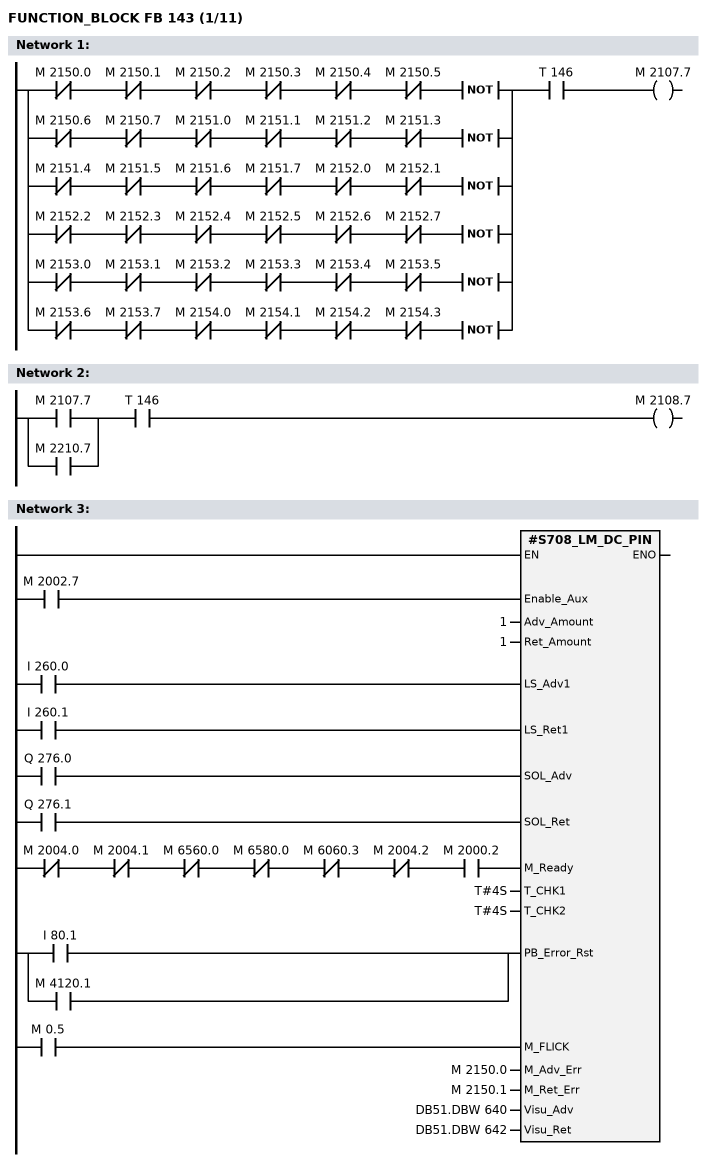

      A(    ;
      AN    M   2150.0;
      AN    M   2150.1;
      AN    M   2150.2;
      AN    M   2150.3;
      AN    M   2150.4;
      AN    M   2150.5;
      NOT   ;
      O(    ;
      AN    M   2150.6;
      AN    M   2150.7;
      AN    M   2151.0;
      AN    M   2151.1;
      AN    M   2151.2;
      AN    M   2151.3;
      NOT   ;
      )     ;
      O(    ;
      AN    M   2151.4;
      AN    M   2151.5;
      AN    M   2151.6;
      AN    M   2151.7;
      AN    M   2152.0;
      AN    M   2152.1;
      NOT   ;
      )     ;
      O(    ;
      AN    M   2152.2;
      AN    M   2152.3;
      AN    M   2152.4;
      AN    M   2152.5;
      AN    M   2152.6;
      AN    M   2152.7;
      NOT   ;
      )     ;
      O(    ;
      AN    M   2153.0;
      AN    M   2153.1;
      AN    M   2153.2;
      AN    M   2153.3;
      AN    M   2153.4;
      AN    M   2153.5;
      NOT   ;
      )     ;
      O(    ;
      AN    M   2153.6;
      AN    M   2153.7;
      AN    M   2154.0;
      AN    M   2154.1;
      AN    M   2154.2;
      AN    M   2154.3;
      NOT   ;
      )     ;
      )     ;
      A     T    146;
      =     M   2107.7;
NETWORK
TITLE =

      A(    ;
      O     M   2107.7;
      O     M   2210.7;
      )     ;
      A     T    146;
      =     M   2108.7;
NETWORK
TITLE =

      A     M   2002.7;
      =     L      0.0;
      BLD   103;
      A     I    260.0;
      =     L      0.1;
      BLD   103;
      A     I    260.1;
      =     L      0.2;
      BLD   103;
      A     Q    276.0;
      =     L      1.1;
      BLD   103;
      A     Q    276.1;
      =     L      1.2;
      BLD   103;
      AN    M   2004.0;
      AN    M   2004.1;
      AN    M   6560.0;
      AN    M   6580.0;
      AN    M   6060.3;
      AN    M   2004.2;
      A     M   2000.2;
      =     L      1.3;
      BLD   103;
      A(    ;
      O     I     80.1;
      O     M   4120.1;
      )     ;
      =     L      1.5;
      BLD   103;
      A     M      0.5;
      =     L      1.6;
      BLD   103;
      CALL #S708_LM_DC_PIN (
           Enable_Aux               := L      0.0,
           Adv_Amount               := 1,
           Ret_Amount               := 1,
           LS_Adv1                  := L      0.1,
           LS_Ret1                  := L      0.2,
           SOL_Adv                  := L      1.1,
           SOL_Ret                  := L      1.2,
           M_Ready                  := L      1.3,
           T_CHK1                   := T#4S,
           T_CHK2                   := T#4S,
           PB_Error_Rst             := L      1.5,
           M_FLICK                  := L      1.6,
           M_Adv_Err                := M   2150.0,
           M_Ret_Err                := M   2150.1,
           Visu_Adv                 := DB51.DBW  640,
           Visu_Ret                 := DB51.DBW  642);
      NOP   0;
NETWORK
TITLE =
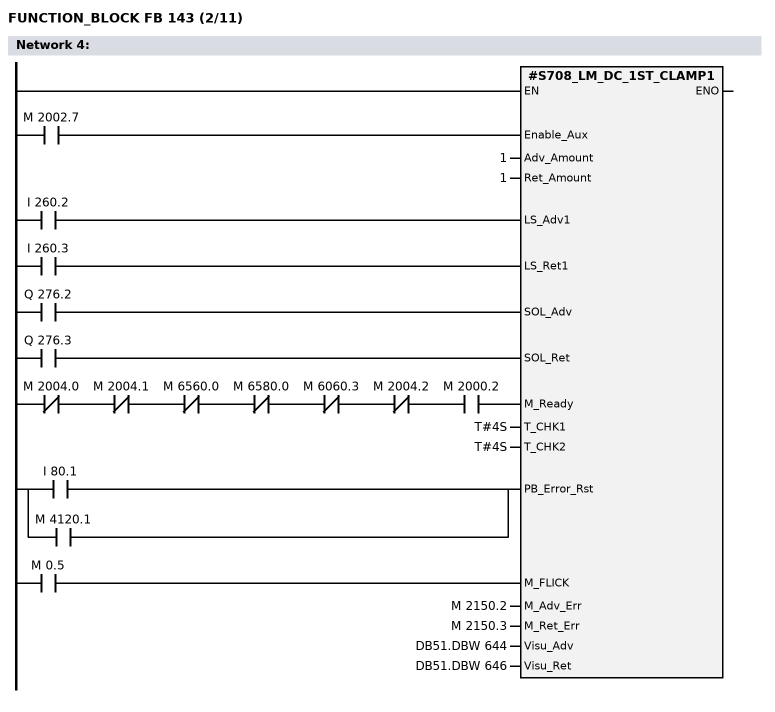

      A     M   2002.7;
      =     L      0.0;
      BLD   103;
      A     I    260.2;
      =     L      0.1;
      BLD   103;
      A     I    260.3;
      =     L      0.2;
      BLD   103;
      A     Q    276.2;
      =     L      1.1;
      BLD   103;
      A     Q    276.3;
      =     L      1.2;
      BLD   103;
      AN    M   2004.0;
      AN    M   2004.1;
      AN    M   6560.0;
      AN    M   6580.0;
      AN    M   6060.3;
      AN    M   2004.2;
      A     M   2000.2;
      =     L      1.3;
      BLD   103;
      A(    ;
      O     I     80.1;
      O     M   4120.1;
      )     ;
      =     L      1.5;
      BLD   103;
      A     M      0.5;
      =     L      1.6;
      BLD   103;
      CALL #S708_LM_DC_1ST_CLAMP1 (
           Enable_Aux               := L      0.0,
           Adv_Amount               := 1,
           Ret_Amount               := 1,
           LS_Adv1                  := L      0.1,
           LS_Ret1                  := L      0.2,
           SOL_Adv                  := L      1.1,
           SOL_Ret                  := L      1.2,
           M_Ready                  := L      1.3,
           T_CHK1                   := T#4S,
           T_CHK2                   := T#4S,
           PB_Error_Rst             := L      1.5,
           M_FLICK                  := L      1.6,
           M_Adv_Err                := M   2150.2,
           M_Ret_Err                := M   2150.3,
           Visu_Adv                 := DB51.DBW  644,
           Visu_Ret                 := DB51.DBW  646);
      NOP   0;
NETWORK
TITLE =
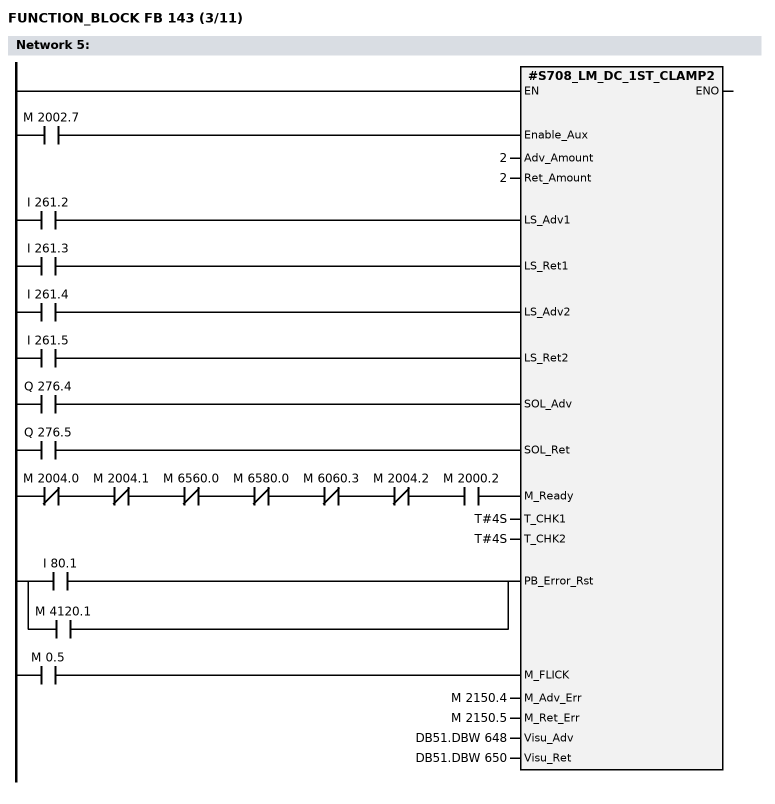

      A     M   2002.7;
      =     L      0.0;
      BLD   103;
      A     I    261.2;
      =     L      0.1;
      BLD   103;
      A     I    261.3;
      =     L      0.2;
      BLD   103;
      A     I    261.4;
      =     L      0.3;
      BLD   103;
      A     I    261.5;
      =     L      0.4;
      BLD   103;
      A     Q    276.4;
      =     L      1.1;
      BLD   103;
      A     Q    276.5;
      =     L      1.2;
      BLD   103;
      AN    M   2004.0;
      AN    M   2004.1;
      AN    M   6560.0;
      AN    M   6580.0;
      AN    M   6060.3;
      AN    M   2004.2;
      A     M   2000.2;
      =     L      1.3;
      BLD   103;
      A(    ;
      O     I     80.1;
      O     M   4120.1;
      )     ;
      =     L      1.5;
      BLD   103;
      A     M      0.5;
      =     L      1.6;
      BLD   103;
      CALL #S708_LM_DC_1ST_CLAMP2 (
           Enable_Aux               := L      0.0,
           Adv_Amount               := 2,
           Ret_Amount               := 2,
           LS_Adv1                  := L      0.1,
           LS_Ret1                  := L      0.2,
           LS_Adv2                  := L      0.3,
           LS_Ret2                  := L      0.4,
           SOL_Adv                  := L      1.1,
           SOL_Ret                  := L      1.2,
           M_Ready                  := L      1.3,
           T_CHK1                   := T#4S,
           T_CHK2                   := T#4S,
           PB_Error_Rst             := L      1.5,
           M_FLICK                  := L      1.6,
           M_Adv_Err                := M   2150.4,
           M_Ret_Err                := M   2150.5,
           Visu_Adv                 := DB51.DBW  648,
           Visu_Ret                 := DB51.DBW  650);
      NOP   0;
NETWORK
TITLE =
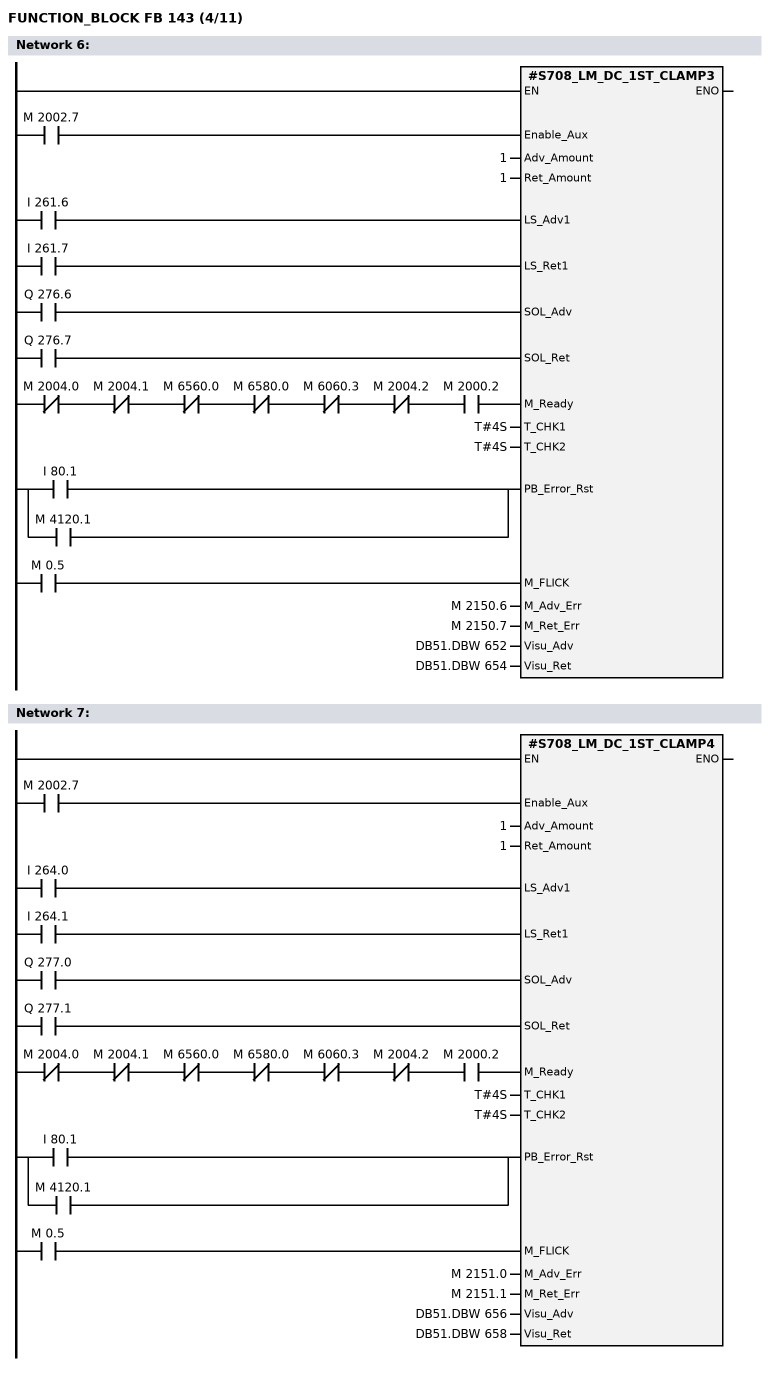

      A     M   2002.7;
      =     L      0.0;
      BLD   103;
      A     I    261.6;
      =     L      0.1;
      BLD   103;
      A     I    261.7;
      =     L      0.2;
      BLD   103;
      A     Q    276.6;
      =     L      1.1;
      BLD   103;
      A     Q    276.7;
      =     L      1.2;
      BLD   103;
      AN    M   2004.0;
      AN    M   2004.1;
      AN    M   6560.0;
      AN    M   6580.0;
      AN    M   6060.3;
      AN    M   2004.2;
      A     M   2000.2;
      =     L      1.3;
      BLD   103;
      A(    ;
      O     I     80.1;
      O     M   4120.1;
      )     ;
      =     L      1.5;
      BLD   103;
      A     M      0.5;
      =     L      1.6;
      BLD   103;
      CALL #S708_LM_DC_1ST_CLAMP3 (
           Enable_Aux               := L      0.0,
           Adv_Amount               := 1,
           Ret_Amount               := 1,
           LS_Adv1                  := L      0.1,
           LS_Ret1                  := L      0.2,
           SOL_Adv                  := L      1.1,
           SOL_Ret                  := L      1.2,
           M_Ready                  := L      1.3,
           T_CHK1                   := T#4S,
           T_CHK2                   := T#4S,
           PB_Error_Rst             := L      1.5,
           M_FLICK                  := L      1.6,
           M_Adv_Err                := M   2150.6,
           M_Ret_Err                := M   2150.7,
           Visu_Adv                 := DB51.DBW  652,
           Visu_Ret                 := DB51.DBW  654);
      NOP   0;
NETWORK
TITLE =

      A     M   2002.7;
      =     L      0.0;
      BLD   103;
      A     I    264.0;
      =     L      0.1;
      BLD   103;
      A     I    264.1;
      =     L      0.2;
      BLD   103;
      A     Q    277.0;
      =     L      1.1;
      BLD   103;
      A     Q    277.1;
      =     L      1.2;
      BLD   103;
      AN    M   2004.0;
      AN    M   2004.1;
      AN    M   6560.0;
      AN    M   6580.0;
      AN    M   6060.3;
      AN    M   2004.2;
      A     M   2000.2;
      =     L      1.3;
      BLD   103;
      A(    ;
      O     I     80.1;
      O     M   4120.1;
      )     ;
      =     L      1.5;
      BLD   103;
      A     M      0.5;
      =     L      1.6;
      BLD   103;
      CALL #S708_LM_DC_1ST_CLAMP4 (
           Enable_Aux               := L      0.0,
           Adv_Amount               := 1,
           Ret_Amount               := 1,
           LS_Adv1                  := L      0.1,
           LS_Ret1                  := L      0.2,
           SOL_Adv                  := L      1.1,
           SOL_Ret                  := L      1.2,
           M_Ready                  := L      1.3,
           T_CHK1                   := T#4S,
           T_CHK2                   := T#4S,
           PB_Error_Rst             := L      1.5,
           M_FLICK                  := L      1.6,
           M_Adv_Err                := M   2151.0,
           M_Ret_Err                := M   2151.1,
           Visu_Adv                 := DB51.DBW  656,
           Visu_Ret                 := DB51.DBW  658);
      NOP   0;
NETWORK
TITLE =
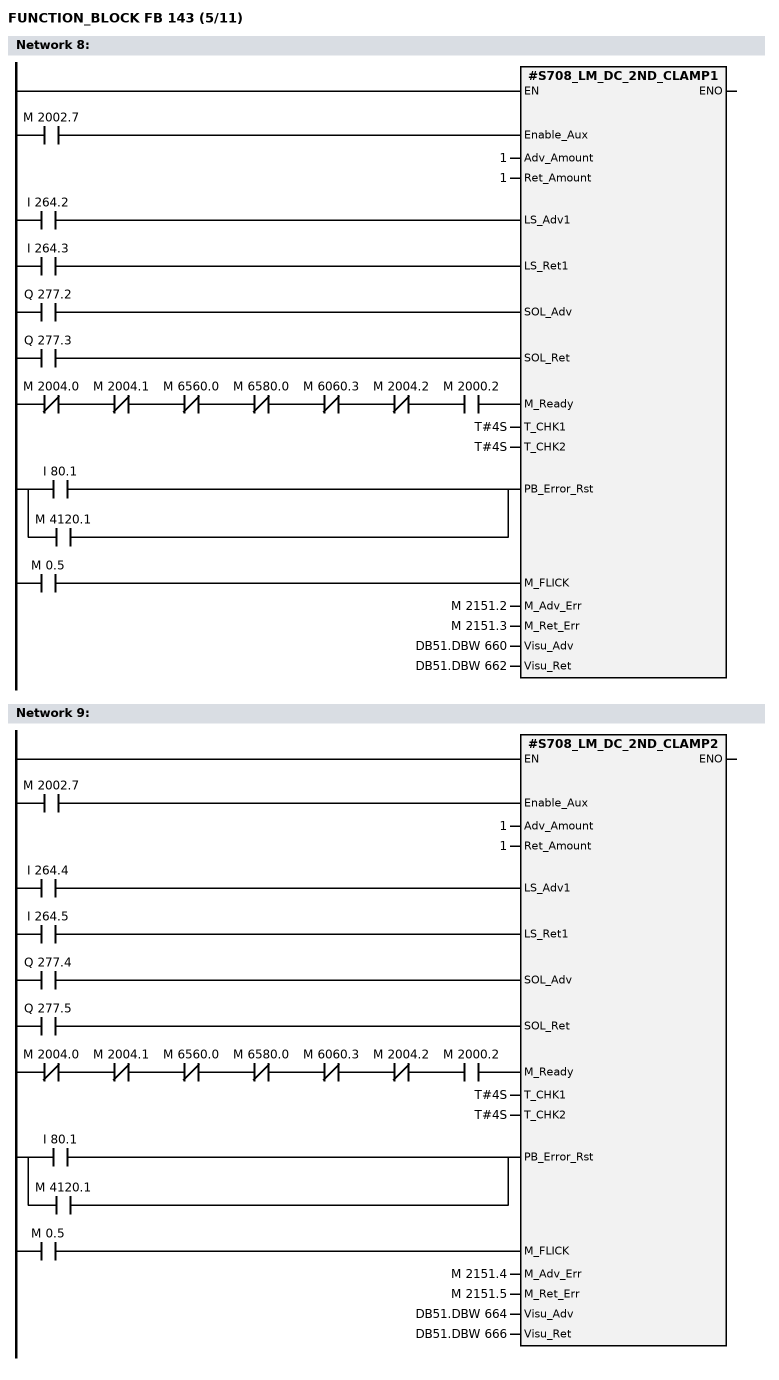

      A     M   2002.7;
      =     L      0.0;
      BLD   103;
      A     I    264.2;
      =     L      0.1;
      BLD   103;
      A     I    264.3;
      =     L      0.2;
      BLD   103;
      A     Q    277.2;
      =     L      1.1;
      BLD   103;
      A     Q    277.3;
      =     L      1.2;
      BLD   103;
      AN    M   2004.0;
      AN    M   2004.1;
      AN    M   6560.0;
      AN    M   6580.0;
      AN    M   6060.3;
      AN    M   2004.2;
      A     M   2000.2;
      =     L      1.3;
      BLD   103;
      A(    ;
      O     I     80.1;
      O     M   4120.1;
      )     ;
      =     L      1.5;
      BLD   103;
      A     M      0.5;
      =     L      1.6;
      BLD   103;
      CALL #S708_LM_DC_2ND_CLAMP1 (
           Enable_Aux               := L      0.0,
           Adv_Amount               := 1,
           Ret_Amount               := 1,
           LS_Adv1                  := L      0.1,
           LS_Ret1                  := L      0.2,
           SOL_Adv                  := L      1.1,
           SOL_Ret                  := L      1.2,
           M_Ready                  := L      1.3,
           T_CHK1                   := T#4S,
           T_CHK2                   := T#4S,
           PB_Error_Rst             := L      1.5,
           M_FLICK                  := L      1.6,
           M_Adv_Err                := M   2151.2,
           M_Ret_Err                := M   2151.3,
           Visu_Adv                 := DB51.DBW  660,
           Visu_Ret                 := DB51.DBW  662);
      NOP   0;
NETWORK
TITLE =

      A     M   2002.7;
      =     L      0.0;
      BLD   103;
      A     I    264.4;
      =     L      0.1;
      BLD   103;
      A     I    264.5;
      =     L      0.2;
      BLD   103;
      A     Q    277.4;
      =     L      1.1;
      BLD   103;
      A     Q    277.5;
      =     L      1.2;
      BLD   103;
      AN    M   2004.0;
      AN    M   2004.1;
      AN    M   6560.0;
      AN    M   6580.0;
      AN    M   6060.3;
      AN    M   2004.2;
      A     M   2000.2;
      =     L      1.3;
      BLD   103;
      A(    ;
      O     I     80.1;
      O     M   4120.1;
      )     ;
      =     L      1.5;
      BLD   103;
      A     M      0.5;
      =     L      1.6;
      BLD   103;
      CALL #S708_LM_DC_2ND_CLAMP2 (
           Enable_Aux               := L      0.0,
           Adv_Amount               := 1,
           Ret_Amount               := 1,
           LS_Adv1                  := L      0.1,
           LS_Ret1                  := L      0.2,
           SOL_Adv                  := L      1.1,
           SOL_Ret                  := L      1.2,
           M_Ready                  := L      1.3,
           T_CHK1                   := T#4S,
           T_CHK2                   := T#4S,
           PB_Error_Rst             := L      1.5,
           M_FLICK                  := L      1.6,
           M_Adv_Err                := M   2151.4,
           M_Ret_Err                := M   2151.5,
           Visu_Adv                 := DB51.DBW  664,
           Visu_Ret                 := DB51.DBW  666);
      NOP   0;
NETWORK
TITLE =
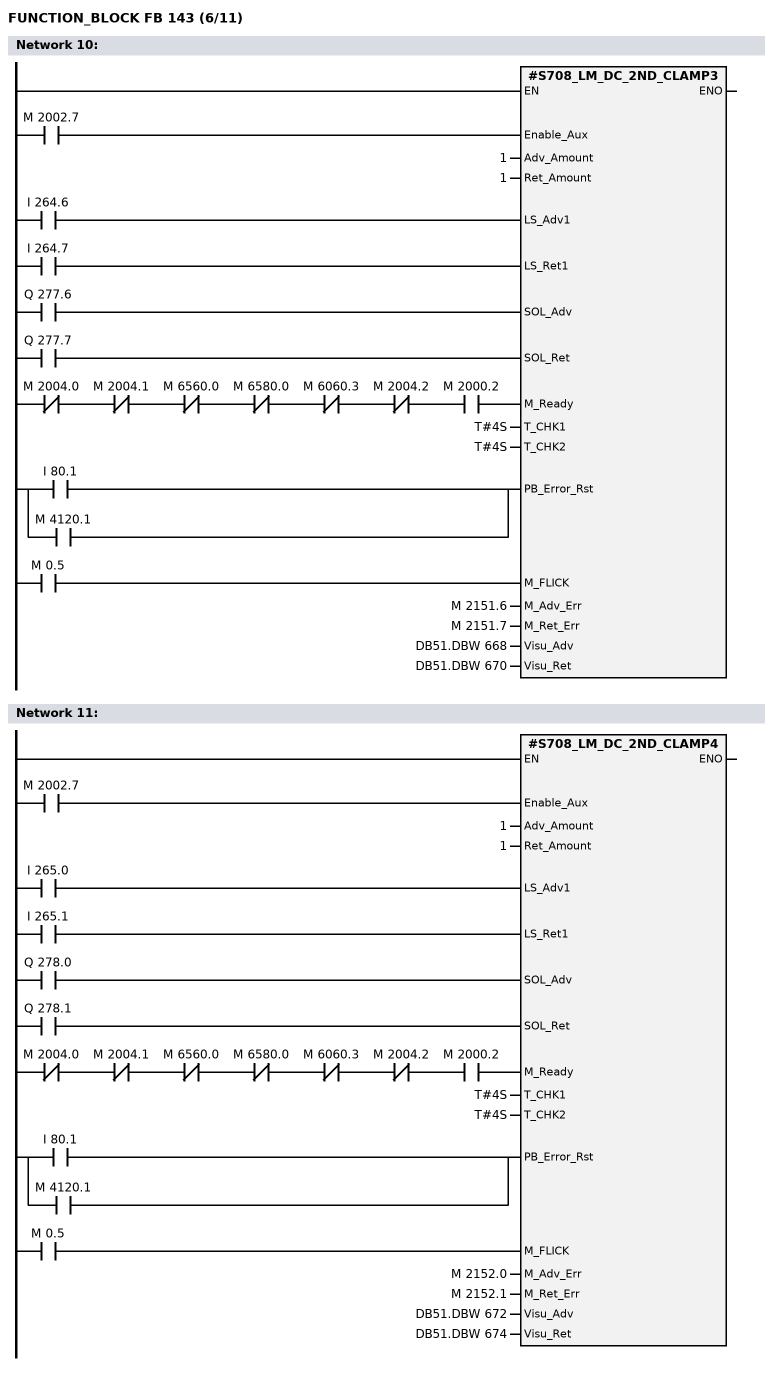

      A     M   2002.7;
      =     L      0.0;
      BLD   103;
      A     I    264.6;
      =     L      0.1;
      BLD   103;
      A     I    264.7;
      =     L      0.2;
      BLD   103;
      A     Q    277.6;
      =     L      1.1;
      BLD   103;
      A     Q    277.7;
      =     L      1.2;
      BLD   103;
      AN    M   2004.0;
      AN    M   2004.1;
      AN    M   6560.0;
      AN    M   6580.0;
      AN    M   6060.3;
      AN    M   2004.2;
      A     M   2000.2;
      =     L      1.3;
      BLD   103;
      A(    ;
      O     I     80.1;
      O     M   4120.1;
      )     ;
      =     L      1.5;
      BLD   103;
      A     M      0.5;
      =     L      1.6;
      BLD   103;
      CALL #S708_LM_DC_2ND_CLAMP3 (
           Enable_Aux               := L      0.0,
           Adv_Amount               := 1,
           Ret_Amount               := 1,
           LS_Adv1                  := L      0.1,
           LS_Ret1                  := L      0.2,
           SOL_Adv                  := L      1.1,
           SOL_Ret                  := L      1.2,
           M_Ready                  := L      1.3,
           T_CHK1                   := T#4S,
           T_CHK2                   := T#4S,
           PB_Error_Rst             := L      1.5,
           M_FLICK                  := L      1.6,
           M_Adv_Err                := M   2151.6,
           M_Ret_Err                := M   2151.7,
           Visu_Adv                 := DB51.DBW  668,
           Visu_Ret                 := DB51.DBW  670);
      NOP   0;
NETWORK
TITLE =

      A     M   2002.7;
      =     L      0.0;
      BLD   103;
      A     I    265.0;
      =     L      0.1;
      BLD   103;
      A     I    265.1;
      =     L      0.2;
      BLD   103;
      A     Q    278.0;
      =     L      1.1;
      BLD   103;
      A     Q    278.1;
      =     L      1.2;
      BLD   103;
      AN    M   2004.0;
      AN    M   2004.1;
      AN    M   6560.0;
      AN    M   6580.0;
      AN    M   6060.3;
      AN    M   2004.2;
      A     M   2000.2;
      =     L      1.3;
      BLD   103;
      A(    ;
      O     I     80.1;
      O     M   4120.1;
      )     ;
      =     L      1.5;
      BLD   103;
      A     M      0.5;
      =     L      1.6;
      BLD   103;
      CALL #S708_LM_DC_2ND_CLAMP4 (
           Enable_Aux               := L      0.0,
           Adv_Amount               := 1,
           Ret_Amount               := 1,
           LS_Adv1                  := L      0.1,
           LS_Ret1                  := L      0.2,
           SOL_Adv                  := L      1.1,
           SOL_Ret                  := L      1.2,
           M_Ready                  := L      1.3,
           T_CHK1                   := T#4S,
           T_CHK2                   := T#4S,
           PB_Error_Rst             := L      1.5,
           M_FLICK                  := L      1.6,
           M_Adv_Err                := M   2152.0,
           M_Ret_Err                := M   2152.1,
           Visu_Adv                 := DB51.DBW  672,
           Visu_Ret                 := DB51.DBW  674);
      NOP   0;
NETWORK
TITLE =
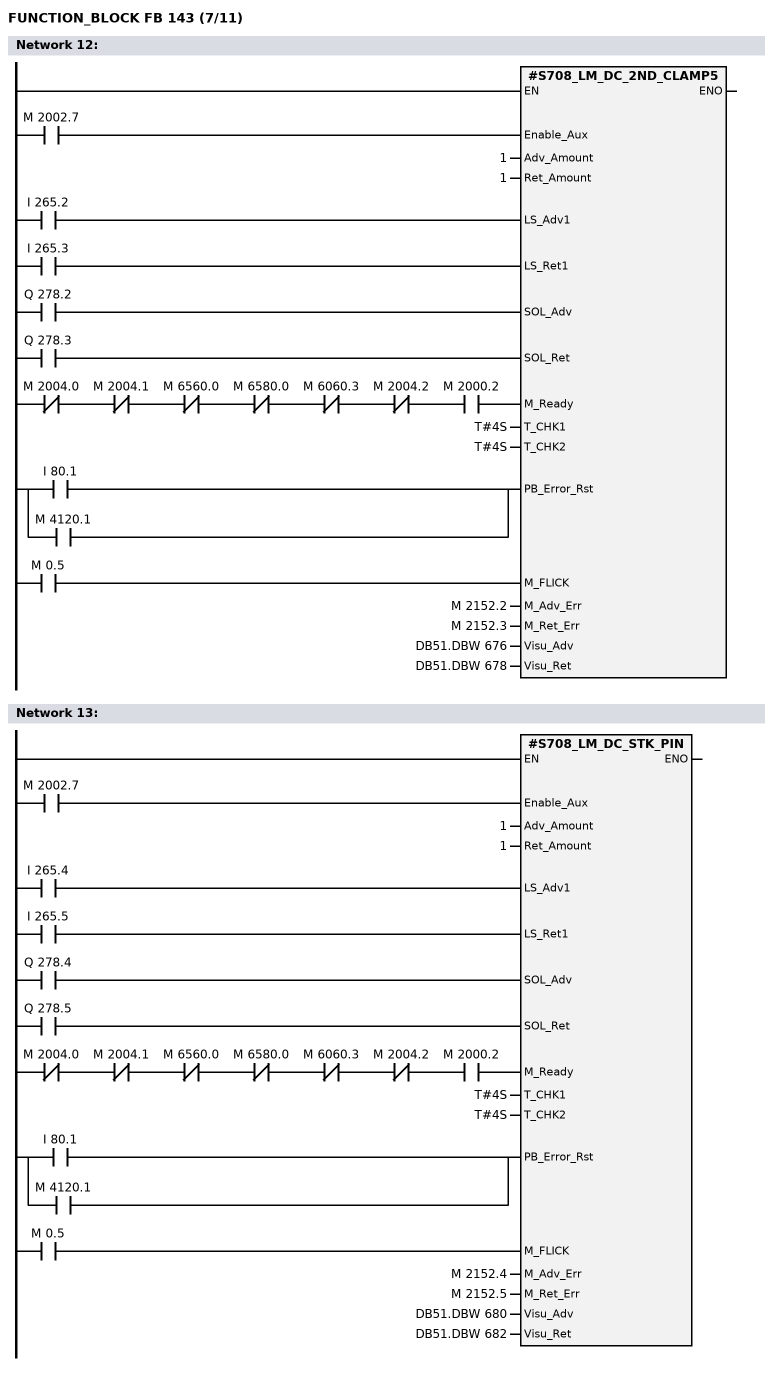

      A     M   2002.7;
      =     L      0.0;
      BLD   103;
      A     I    265.2;
      =     L      0.1;
      BLD   103;
      A     I    265.3;
      =     L      0.2;
      BLD   103;
      A     Q    278.2;
      =     L      1.1;
      BLD   103;
      A     Q    278.3;
      =     L      1.2;
      BLD   103;
      AN    M   2004.0;
      AN    M   2004.1;
      AN    M   6560.0;
      AN    M   6580.0;
      AN    M   6060.3;
      AN    M   2004.2;
      A     M   2000.2;
      =     L      1.3;
      BLD   103;
      A(    ;
      O     I     80.1;
      O     M   4120.1;
      )     ;
      =     L      1.5;
      BLD   103;
      A     M      0.5;
      =     L      1.6;
      BLD   103;
      CALL #S708_LM_DC_2ND_CLAMP5 (
           Enable_Aux               := L      0.0,
           Adv_Amount               := 1,
           Ret_Amount               := 1,
           LS_Adv1                  := L      0.1,
           LS_Ret1                  := L      0.2,
           SOL_Adv                  := L      1.1,
           SOL_Ret                  := L      1.2,
           M_Ready                  := L      1.3,
           T_CHK1                   := T#4S,
           T_CHK2                   := T#4S,
           PB_Error_Rst             := L      1.5,
           M_FLICK                  := L      1.6,
           M_Adv_Err                := M   2152.2,
           M_Ret_Err                := M   2152.3,
           Visu_Adv                 := DB51.DBW  676,
           Visu_Ret                 := DB51.DBW  678);
      NOP   0;
NETWORK
TITLE =

      A     M   2002.7;
      =     L      0.0;
      BLD   103;
      A     I    265.4;
      =     L      0.1;
      BLD   103;
      A     I    265.5;
      =     L      0.2;
      BLD   103;
      A     Q    278.4;
      =     L      1.1;
      BLD   103;
      A     Q    278.5;
      =     L      1.2;
      BLD   103;
      AN    M   2004.0;
      AN    M   2004.1;
      AN    M   6560.0;
      AN    M   6580.0;
      AN    M   6060.3;
      AN    M   2004.2;
      A     M   2000.2;
      =     L      1.3;
      BLD   103;
      A(    ;
      O     I     80.1;
      O     M   4120.1;
      )     ;
      =     L      1.5;
      BLD   103;
      A     M      0.5;
      =     L      1.6;
      BLD   103;
      CALL #S708_LM_DC_STK_PIN (
           Enable_Aux               := L      0.0,
           Adv_Amount               := 1,
           Ret_Amount               := 1,
           LS_Adv1                  := L      0.1,
           LS_Ret1                  := L      0.2,
           SOL_Adv                  := L      1.1,
           SOL_Ret                  := L      1.2,
           M_Ready                  := L      1.3,
           T_CHK1                   := T#4S,
           T_CHK2                   := T#4S,
           PB_Error_Rst             := L      1.5,
           M_FLICK                  := L      1.6,
           M_Adv_Err                := M   2152.4,
           M_Ret_Err                := M   2152.5,
           Visu_Adv                 := DB51.DBW  680,
           Visu_Ret                 := DB51.DBW  682);
      NOP   0;
NETWORK
TITLE =
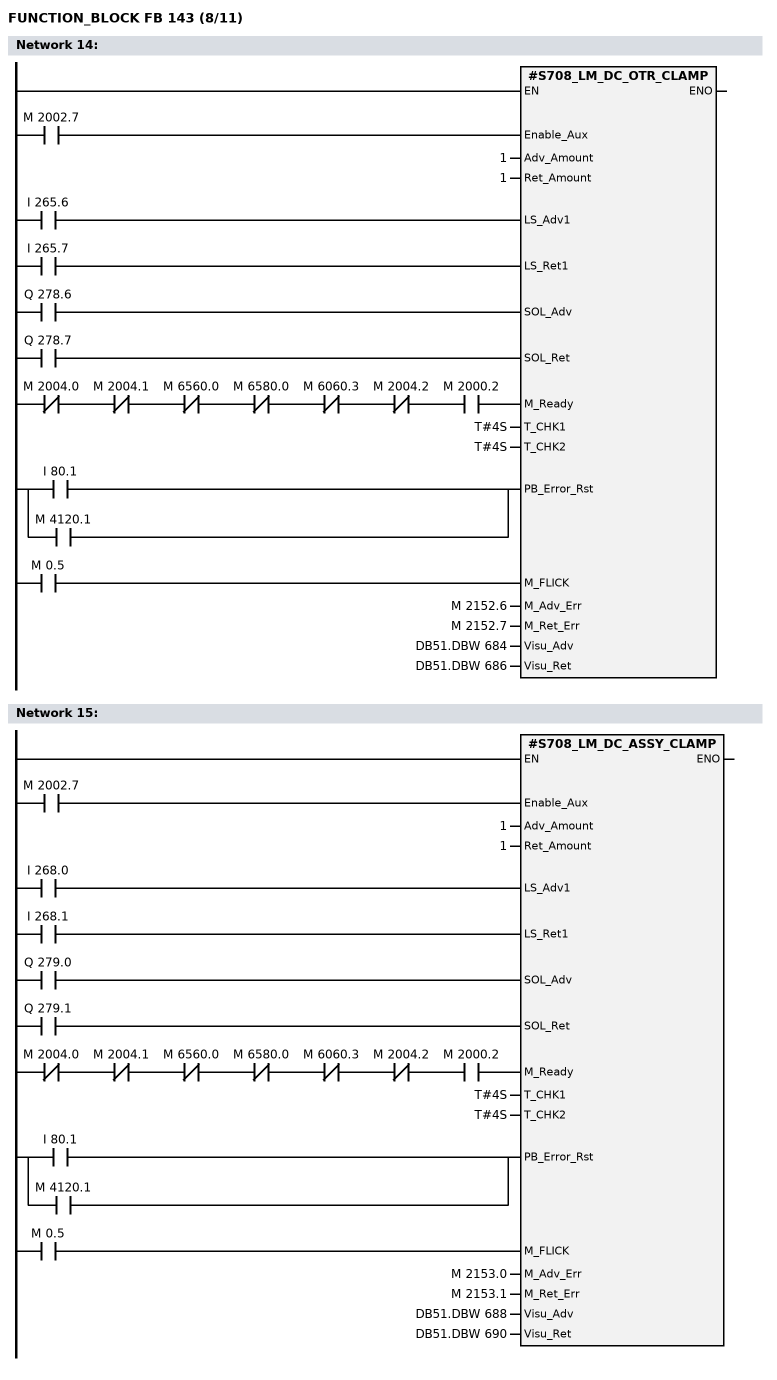

      A     M   2002.7;
      =     L      0.0;
      BLD   103;
      A     I    265.6;
      =     L      0.1;
      BLD   103;
      A     I    265.7;
      =     L      0.2;
      BLD   103;
      A     Q    278.6;
      =     L      1.1;
      BLD   103;
      A     Q    278.7;
      =     L      1.2;
      BLD   103;
      AN    M   2004.0;
      AN    M   2004.1;
      AN    M   6560.0;
      AN    M   6580.0;
      AN    M   6060.3;
      AN    M   2004.2;
      A     M   2000.2;
      =     L      1.3;
      BLD   103;
      A(    ;
      O     I     80.1;
      O     M   4120.1;
      )     ;
      =     L      1.5;
      BLD   103;
      A     M      0.5;
      =     L      1.6;
      BLD   103;
      CALL #S708_LM_DC_OTR_CLAMP (
           Enable_Aux               := L      0.0,
           Adv_Amount               := 1,
           Ret_Amount               := 1,
           LS_Adv1                  := L      0.1,
           LS_Ret1                  := L      0.2,
           SOL_Adv                  := L      1.1,
           SOL_Ret                  := L      1.2,
           M_Ready                  := L      1.3,
           T_CHK1                   := T#4S,
           T_CHK2                   := T#4S,
           PB_Error_Rst             := L      1.5,
           M_FLICK                  := L      1.6,
           M_Adv_Err                := M   2152.6,
           M_Ret_Err                := M   2152.7,
           Visu_Adv                 := DB51.DBW  684,
           Visu_Ret                 := DB51.DBW  686);
      NOP   0;
NETWORK
TITLE =

      A     M   2002.7;
      =     L      0.0;
      BLD   103;
      A     I    268.0;
      =     L      0.1;
      BLD   103;
      A     I    268.1;
      =     L      0.2;
      BLD   103;
      A     Q    279.0;
      =     L      1.1;
      BLD   103;
      A     Q    279.1;
      =     L      1.2;
      BLD   103;
      AN    M   2004.0;
      AN    M   2004.1;
      AN    M   6560.0;
      AN    M   6580.0;
      AN    M   6060.3;
      AN    M   2004.2;
      A     M   2000.2;
      =     L      1.3;
      BLD   103;
      A(    ;
      O     I     80.1;
      O     M   4120.1;
      )     ;
      =     L      1.5;
      BLD   103;
      A     M      0.5;
      =     L      1.6;
      BLD   103;
      CALL #S708_LM_DC_ASSY_CLAMP (
           Enable_Aux               := L      0.0,
           Adv_Amount               := 1,
           Ret_Amount               := 1,
           LS_Adv1                  := L      0.1,
           LS_Ret1                  := L      0.2,
           SOL_Adv                  := L      1.1,
           SOL_Ret                  := L      1.2,
           M_Ready                  := L      1.3,
           T_CHK1                   := T#4S,
           T_CHK2                   := T#4S,
           PB_Error_Rst             := L      1.5,
           M_FLICK                  := L      1.6,
           M_Adv_Err                := M   2153.0,
           M_Ret_Err                := M   2153.1,
           Visu_Adv                 := DB51.DBW  688,
           Visu_Ret                 := DB51.DBW  690);
      NOP   0;
NETWORK
TITLE =
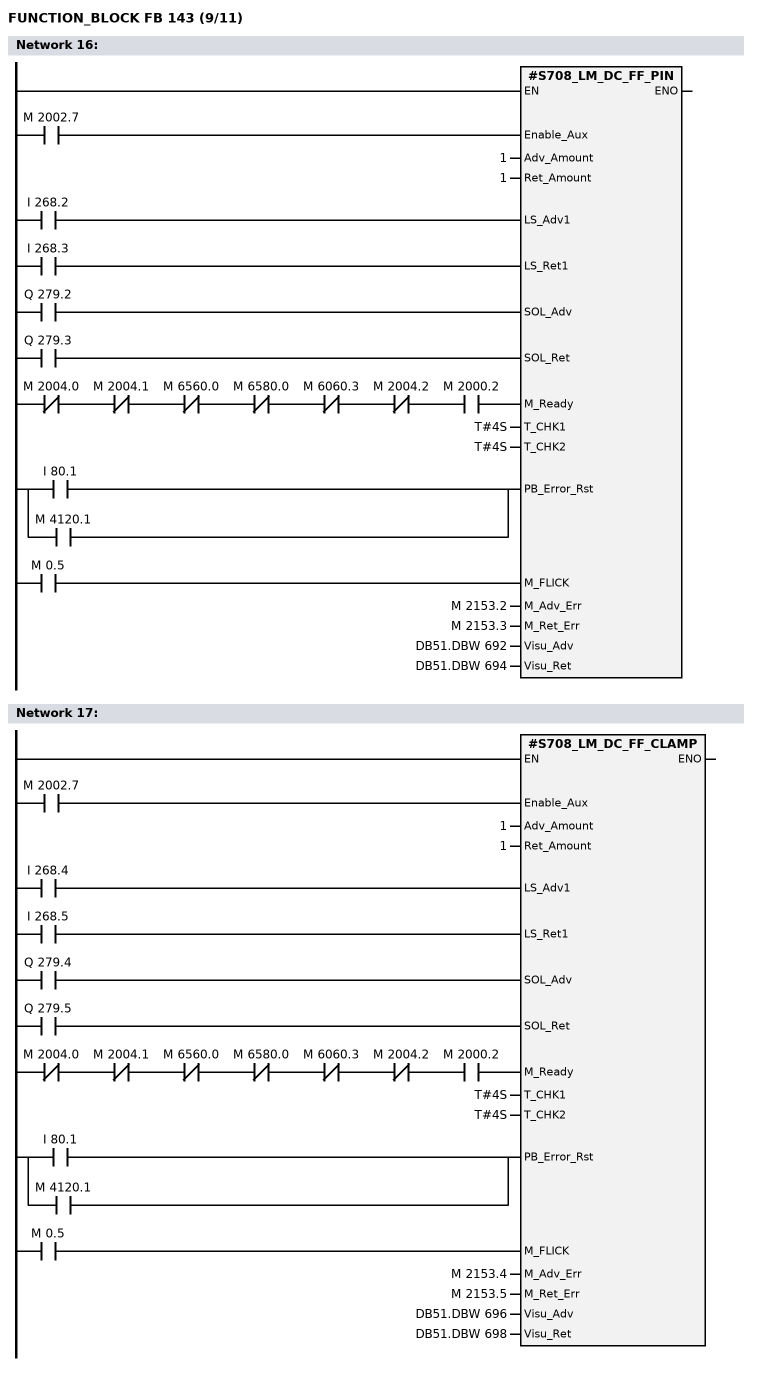

      A     M   2002.7;
      =     L      0.0;
      BLD   103;
      A     I    268.2;
      =     L      0.1;
      BLD   103;
      A     I    268.3;
      =     L      0.2;
      BLD   103;
      A     Q    279.2;
      =     L      1.1;
      BLD   103;
      A     Q    279.3;
      =     L      1.2;
      BLD   103;
      AN    M   2004.0;
      AN    M   2004.1;
      AN    M   6560.0;
      AN    M   6580.0;
      AN    M   6060.3;
      AN    M   2004.2;
      A     M   2000.2;
      =     L      1.3;
      BLD   103;
      A(    ;
      O     I     80.1;
      O     M   4120.1;
      )     ;
      =     L      1.5;
      BLD   103;
      A     M      0.5;
      =     L      1.6;
      BLD   103;
      CALL #S708_LM_DC_FF_PIN (
           Enable_Aux               := L      0.0,
           Adv_Amount               := 1,
           Ret_Amount               := 1,
           LS_Adv1                  := L      0.1,
           LS_Ret1                  := L      0.2,
           SOL_Adv                  := L      1.1,
           SOL_Ret                  := L      1.2,
           M_Ready                  := L      1.3,
           T_CHK1                   := T#4S,
           T_CHK2                   := T#4S,
           PB_Error_Rst             := L      1.5,
           M_FLICK                  := L      1.6,
           M_Adv_Err                := M   2153.2,
           M_Ret_Err                := M   2153.3,
           Visu_Adv                 := DB51.DBW  692,
           Visu_Ret                 := DB51.DBW  694);
      NOP   0;
NETWORK
TITLE =

      A     M   2002.7;
      =     L      0.0;
      BLD   103;
      A     I    268.4;
      =     L      0.1;
      BLD   103;
      A     I    268.5;
      =     L      0.2;
      BLD   103;
      A     Q    279.4;
      =     L      1.1;
      BLD   103;
      A     Q    279.5;
      =     L      1.2;
      BLD   103;
      AN    M   2004.0;
      AN    M   2004.1;
      AN    M   6560.0;
      AN    M   6580.0;
      AN    M   6060.3;
      AN    M   2004.2;
      A     M   2000.2;
      =     L      1.3;
      BLD   103;
      A(    ;
      O     I     80.1;
      O     M   4120.1;
      )     ;
      =     L      1.5;
      BLD   103;
      A     M      0.5;
      =     L      1.6;
      BLD   103;
      CALL #S708_LM_DC_FF_CLAMP (
           Enable_Aux               := L      0.0,
           Adv_Amount               := 1,
           Ret_Amount               := 1,
           LS_Adv1                  := L      0.1,
           LS_Ret1                  := L      0.2,
           SOL_Adv                  := L      1.1,
           SOL_Ret                  := L      1.2,
           M_Ready                  := L      1.3,
           T_CHK1                   := T#4S,
           T_CHK2                   := T#4S,
           PB_Error_Rst             := L      1.5,
           M_FLICK                  := L      1.6,
           M_Adv_Err                := M   2153.4,
           M_Ret_Err                := M   2153.5,
           Visu_Adv                 := DB51.DBW  696,
           Visu_Ret                 := DB51.DBW  698);
      NOP   0;
NETWORK
TITLE =
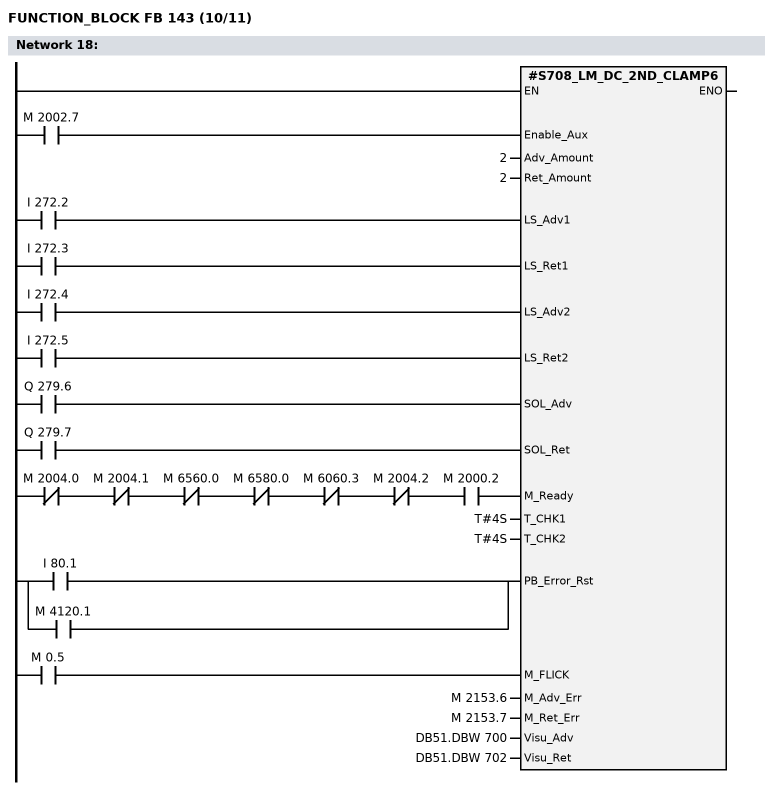

      A     M   2002.7;
      =     L      0.0;
      BLD   103;
      A     I    272.2;
      =     L      0.1;
      BLD   103;
      A     I    272.3;
      =     L      0.2;
      BLD   103;
      A     I    272.4;
      =     L      0.3;
      BLD   103;
      A     I    272.5;
      =     L      0.4;
      BLD   103;
      A     Q    279.6;
      =     L      1.1;
      BLD   103;
      A     Q    279.7;
      =     L      1.2;
      BLD   103;
      AN    M   2004.0;
      AN    M   2004.1;
      AN    M   6560.0;
      AN    M   6580.0;
      AN    M   6060.3;
      AN    M   2004.2;
      A     M   2000.2;
      =     L      1.3;
      BLD   103;
      A(    ;
      O     I     80.1;
      O     M   4120.1;
      )     ;
      =     L      1.5;
      BLD   103;
      A     M      0.5;
      =     L      1.6;
      BLD   103;
      CALL #S708_LM_DC_2ND_CLAMP6 (
           Enable_Aux               := L      0.0,
           Adv_Amount               := 2,
           Ret_Amount               := 2,
           LS_Adv1                  := L      0.1,
           LS_Ret1                  := L      0.2,
           LS_Adv2                  := L      0.3,
           LS_Ret2                  := L      0.4,
           SOL_Adv                  := L      1.1,
           SOL_Ret                  := L      1.2,
           M_Ready                  := L      1.3,
           T_CHK1                   := T#4S,
           T_CHK2                   := T#4S,
           PB_Error_Rst             := L      1.5,
           M_FLICK                  := L      1.6,
           M_Adv_Err                := M   2153.6,
           M_Ret_Err                := M   2153.7,
           Visu_Adv                 := DB51.DBW  700,
           Visu_Ret                 := DB51.DBW  702);
      NOP   0;
NETWORK
TITLE =
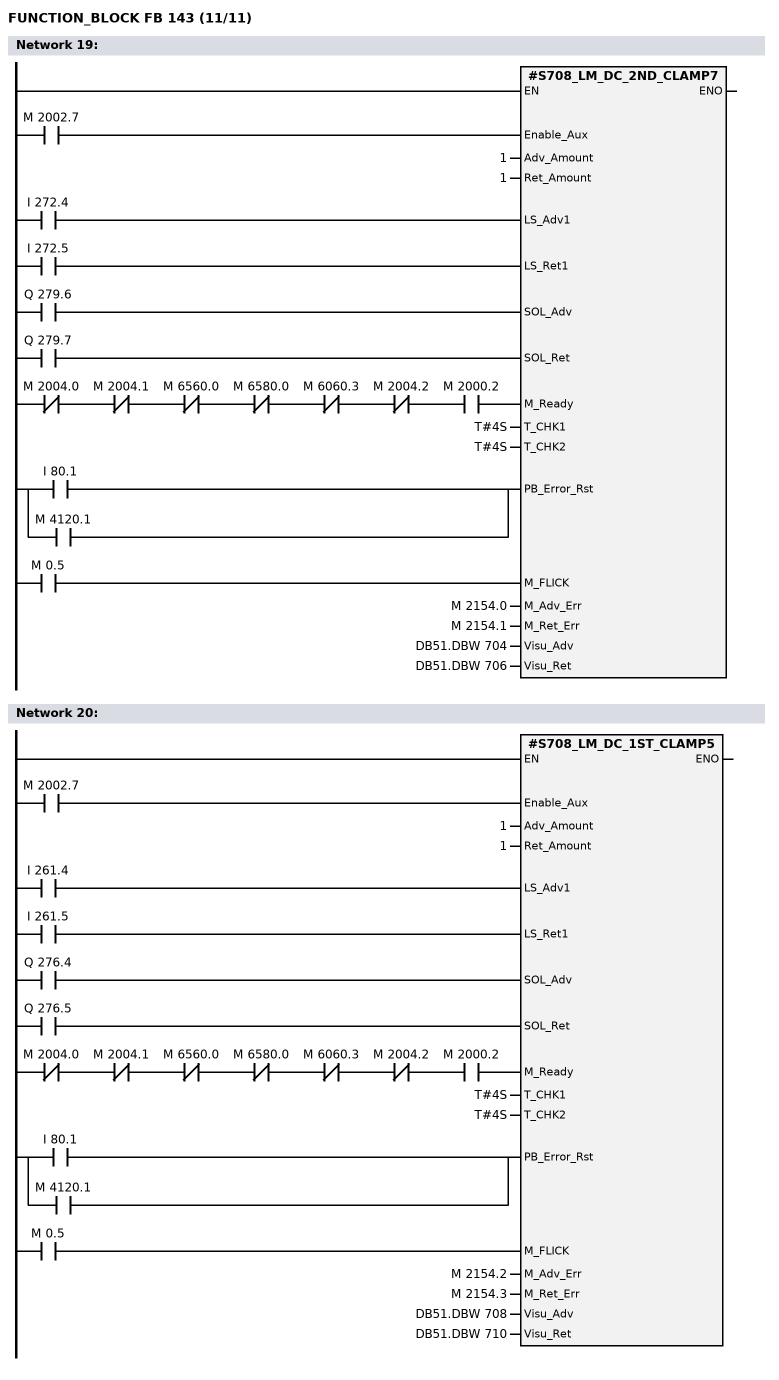

      A     M   2002.7;
      =     L      0.0;
      BLD   103;
      A     I    272.4;
      =     L      0.1;
      BLD   103;
      A     I    272.5;
      =     L      0.2;
      BLD   103;
      A     Q    279.6;
      =     L      1.1;
      BLD   103;
      A     Q    279.7;
      =     L      1.2;
      BLD   103;
      AN    M   2004.0;
      AN    M   2004.1;
      AN    M   6560.0;
      AN    M   6580.0;
      AN    M   6060.3;
      AN    M   2004.2;
      A     M   2000.2;
      =     L      1.3;
      BLD   103;
      A(    ;
      O     I     80.1;
      O     M   4120.1;
      )     ;
      =     L      1.5;
      BLD   103;
      A     M      0.5;
      =     L      1.6;
      BLD   103;
      CALL #S708_LM_DC_2ND_CLAMP7 (
           Enable_Aux               := L      0.0,
           Adv_Amount               := 1,
           Ret_Amount               := 1,
           LS_Adv1                  := L      0.1,
           LS_Ret1                  := L      0.2,
           SOL_Adv                  := L      1.1,
           SOL_Ret                  := L      1.2,
           M_Ready                  := L      1.3,
           T_CHK1                   := T#4S,
           T_CHK2                   := T#4S,
           PB_Error_Rst             := L      1.5,
           M_FLICK                  := L      1.6,
           M_Adv_Err                := M   2154.0,
           M_Ret_Err                := M   2154.1,
           Visu_Adv                 := DB51.DBW  704,
           Visu_Ret                 := DB51.DBW  706);
      NOP   0;
NETWORK
TITLE =

      A     M   2002.7;
      =     L      0.0;
      BLD   103;
      A     I    261.4;
      =     L      0.1;
      BLD   103;
      A     I    261.5;
      =     L      0.2;
      BLD   103;
      A     Q    276.4;
      =     L      1.1;
      BLD   103;
      A     Q    276.5;
      =     L      1.2;
      BLD   103;
      AN    M   2004.0;
      AN    M   2004.1;
      AN    M   6560.0;
      AN    M   6580.0;
      AN    M   6060.3;
      AN    M   2004.2;
      A     M   2000.2;
      =     L      1.3;
      BLD   103;
      A(    ;
      O     I     80.1;
      O     M   4120.1;
      )     ;
      =     L      1.5;
      BLD   103;
      A     M      0.5;
      =     L      1.6;
      BLD   103;
      CALL #S708_LM_DC_1ST_CLAMP5 (
           Enable_Aux               := L      0.0,
           Adv_Amount               := 1,
           Ret_Amount               := 1,
           LS_Adv1                  := L      0.1,
           LS_Ret1                  := L      0.2,
           SOL_Adv                  := L      1.1,
           SOL_Ret                  := L      1.2,
           M_Ready                  := L      1.3,
           T_CHK1                   := T#4S,
           T_CHK2                   := T#4S,
           PB_Error_Rst             := L      1.5,
           M_FLICK                  := L      1.6,
           M_Adv_Err                := M   2154.2,
           M_Ret_Err                := M   2154.3,
           Visu_Adv                 := DB51.DBW  708,
           Visu_Ret                 := DB51.DBW  710);
      NOP   0;
END_FUNCTION_BLOCK

DATA_BLOCK DB 143
TITLE =
VERSION : 0.0

 FB 143
BEGIN
   S708_LM_DC_PIN.Enable_Aux := FALSE;
   S708_LM_DC_PIN.Adv_Amount := 1;
   S708_LM_DC_PIN.Ret_Amount := 1;
   S708_LM_DC_PIN.LS_Adv1 := FALSE;
   S708_LM_DC_PIN.LS_Ret1 := FALSE;
   S708_LM_DC_PIN.LS_Adv2 := FALSE;
   S708_LM_DC_PIN.LS_Ret2 := FALSE;
   S708_LM_DC_PIN.LS_Adv3 := FALSE;
   S708_LM_DC_PIN.LS_Ret3 := FALSE;
   S708_LM_DC_PIN.LS_Adv4 := FALSE;
   S708_LM_DC_PIN.LS_Ret4 := FALSE;
   S708_LM_DC_PIN.SOL_Adv := FALSE;
   S708_LM_DC_PIN.SOL_Ret := FALSE;
   S708_LM_DC_PIN.M_Ready := TRUE;
   S708_LM_DC_PIN.T_CHK1 := T#4S;
   S708_LM_DC_PIN.T_CHK2 := T#4S;
   S708_LM_DC_PIN.PB_Lamp_CHK := FALSE;
   S708_LM_DC_PIN.PB_Error_Rst := FALSE;
   S708_LM_DC_PIN.M_FLICK := FALSE;
   S708_LM_DC_PIN.M_Adv_Err := FALSE;
   S708_LM_DC_PIN.M_Ret_Err := FALSE;
   S708_LM_DC_PIN.LP_Adv := FALSE;
   S708_LM_DC_PIN.LP_Ret := FALSE;
   S708_LM_DC_PIN.Visu_Adv := W#16#0;
   S708_LM_DC_PIN.Visu_Ret := W#16#0;
   S708_LM_DC_PIN.Error_T1.IN := FALSE;
   S708_LM_DC_PIN.Error_T1.PT := T#4S;
   S708_LM_DC_PIN.Error_T1.Q := FALSE;
   S708_LM_DC_PIN.Error_T1.ET := T#0MS;
   S708_LM_DC_PIN.Error_T1.STATE := B#16#0;
   S708_LM_DC_PIN.Error_T1.STIME := T#22D23H1M2S540MS;
   S708_LM_DC_PIN.Error_T1.ATIME := T#22D23H1M4S284MS;
   S708_LM_DC_PIN.Error_T2.IN := FALSE;
   S708_LM_DC_PIN.Error_T2.PT := T#4S;
   S708_LM_DC_PIN.Error_T2.Q := FALSE;
   S708_LM_DC_PIN.Error_T2.ET := T#0MS;
   S708_LM_DC_PIN.Error_T2.STATE := B#16#0;
   S708_LM_DC_PIN.Error_T2.STIME := T#0MS;
   S708_LM_DC_PIN.Error_T2.ATIME := T#0MS;
   S708_LM_DC_PIN.CHK_Aux1 := FALSE;
   S708_LM_DC_PIN.CHK_Aux2 := FALSE;
   S708_LM_DC_PIN.Error_T1_DN := FALSE;
   S708_LM_DC_PIN.Error_T2_DN := FALSE;
   S708_LM_DC_PIN.Adv_Memo := FALSE;
   S708_LM_DC_PIN.Visu_Adv_Arr[0] := FALSE;
   S708_LM_DC_PIN.Visu_Adv_Arr[1] := FALSE;
   S708_LM_DC_PIN.Visu_Adv_Arr[2] := FALSE;
   S708_LM_DC_PIN.Visu_Adv_Arr[3] := FALSE;
   S708_LM_DC_PIN.Visu_Adv_Arr[4] := FALSE;
   S708_LM_DC_PIN.Visu_Adv_Arr[5] := FALSE;
   S708_LM_DC_PIN.Visu_Adv_Arr[6] := FALSE;
   S708_LM_DC_PIN.Visu_Adv_Arr[7] := FALSE;
   S708_LM_DC_PIN.Visu_Adv_Arr[8] := FALSE;
   S708_LM_DC_PIN.Visu_Adv_Arr[9] := FALSE;
   S708_LM_DC_PIN.Visu_Adv_Arr[10] := FALSE;
   S708_LM_DC_PIN.Visu_Adv_Arr[11] := FALSE;
   S708_LM_DC_PIN.Visu_Adv_Arr[12] := FALSE;
   S708_LM_DC_PIN.Visu_Adv_Arr[13] := FALSE;
   S708_LM_DC_PIN.Visu_Adv_Arr[14] := FALSE;
   S708_LM_DC_PIN.Visu_Adv_Arr[15] := FALSE;
   S708_LM_DC_PIN.Visu_Ret_Arr[0] := FALSE;
   S708_LM_DC_PIN.Visu_Ret_Arr[1] := FALSE;
   S708_LM_DC_PIN.Visu_Ret_Arr[2] := FALSE;
   S708_LM_DC_PIN.Visu_Ret_Arr[3] := FALSE;
   S708_LM_DC_PIN.Visu_Ret_Arr[4] := FALSE;
   S708_LM_DC_PIN.Visu_Ret_Arr[5] := FALSE;
   S708_LM_DC_PIN.Visu_Ret_Arr[6] := FALSE;
   S708_LM_DC_PIN.Visu_Ret_Arr[7] := FALSE;
   S708_LM_DC_PIN.Visu_Ret_Arr[8] := FALSE;
   S708_LM_DC_PIN.Visu_Ret_Arr[9] := FALSE;
   S708_LM_DC_PIN.Visu_Ret_Arr[10] := FALSE;
   S708_LM_DC_PIN.Visu_Ret_Arr[11] := FALSE;
   S708_LM_DC_PIN.Visu_Ret_Arr[12] := FALSE;
   S708_LM_DC_PIN.Visu_Ret_Arr[13] := FALSE;
   S708_LM_DC_PIN.Visu_Ret_Arr[14] := FALSE;
   S708_LM_DC_PIN.Visu_Ret_Arr[15] := FALSE;
   S708_LM_DC_PIN.BLK_Move_Ret := 0;
   S708_LM_DC_PIN.Enable := FALSE;
   S708_LM_DC_PIN.Adv_End := FALSE;
   S708_LM_DC_PIN.Ret_End := FALSE;
   S708_LM_DC_1ST_CLAMP1.Enable_Aux := FALSE;
   S708_LM_DC_1ST_CLAMP1.Adv_Amount := 1;
   S708_LM_DC_1ST_CLAMP1.Ret_Amount := 1;
   S708_LM_DC_1ST_CLAMP1.LS_Adv1 := FALSE;
   S708_LM_DC_1ST_CLAMP1.LS_Ret1 := FALSE;
   S708_LM_DC_1ST_CLAMP1.LS_Adv2 := FALSE;
   S708_LM_DC_1ST_CLAMP1.LS_Ret2 := FALSE;
   S708_LM_DC_1ST_CLAMP1.LS_Adv3 := FALSE;
   S708_LM_DC_1ST_CLAMP1.LS_Ret3 := FALSE;
   S708_LM_DC_1ST_CLAMP1.LS_Adv4 := FALSE;
   S708_LM_DC_1ST_CLAMP1.LS_Ret4 := FALSE;
   S708_LM_DC_1ST_CLAMP1.SOL_Adv := FALSE;
   S708_LM_DC_1ST_CLAMP1.SOL_Ret := FALSE;
   S708_LM_DC_1ST_CLAMP1.M_Ready := TRUE;
   S708_LM_DC_1ST_CLAMP1.T_CHK1 := T#4S;
   S708_LM_DC_1ST_CLAMP1.T_CHK2 := T#4S;
   S708_LM_DC_1ST_CLAMP1.PB_Lamp_CHK := FALSE;
   S708_LM_DC_1ST_CLAMP1.PB_Error_Rst := FALSE;
   S708_LM_DC_1ST_CLAMP1.M_FLICK := FALSE;
   S708_LM_DC_1ST_CLAMP1.M_Adv_Err := FALSE;
   S708_LM_DC_1ST_CLAMP1.M_Ret_Err := FALSE;
   S708_LM_DC_1ST_CLAMP1.LP_Adv := FALSE;
   S708_LM_DC_1ST_CLAMP1.LP_Ret := FALSE;
   S708_LM_DC_1ST_CLAMP1.Visu_Adv := W#16#0;
   S708_LM_DC_1ST_CLAMP1.Visu_Ret := W#16#0;
   S708_LM_DC_1ST_CLAMP1.Error_T1.IN := FALSE;
   S708_LM_DC_1ST_CLAMP1.Error_T1.PT := T#4S;
   S708_LM_DC_1ST_CLAMP1.Error_T1.Q := FALSE;
   S708_LM_DC_1ST_CLAMP1.Error_T1.ET := T#0MS;
   S708_LM_DC_1ST_CLAMP1.Error_T1.STATE := B#16#0;
   S708_LM_DC_1ST_CLAMP1.Error_T1.STIME := T#22D23H1M2S540MS;
   S708_LM_DC_1ST_CLAMP1.Error_T1.ATIME := T#22D23H1M3S651MS;
   S708_LM_DC_1ST_CLAMP1.Error_T2.IN := FALSE;
   S708_LM_DC_1ST_CLAMP1.Error_T2.PT := T#4S;
   S708_LM_DC_1ST_CLAMP1.Error_T2.Q := FALSE;
   S708_LM_DC_1ST_CLAMP1.Error_T2.ET := T#0MS;
   S708_LM_DC_1ST_CLAMP1.Error_T2.STATE := B#16#0;
   S708_LM_DC_1ST_CLAMP1.Error_T2.STIME := T#0MS;
   S708_LM_DC_1ST_CLAMP1.Error_T2.ATIME := T#0MS;
   S708_LM_DC_1ST_CLAMP1.CHK_Aux1 := FALSE;
   S708_LM_DC_1ST_CLAMP1.CHK_Aux2 := FALSE;
   S708_LM_DC_1ST_CLAMP1.Error_T1_DN := FALSE;
   S708_LM_DC_1ST_CLAMP1.Error_T2_DN := FALSE;
   S708_LM_DC_1ST_CLAMP1.Adv_Memo := FALSE;
   S708_LM_DC_1ST_CLAMP1.Visu_Adv_Arr[0] := FALSE;
   S708_LM_DC_1ST_CLAMP1.Visu_Adv_Arr[1] := FALSE;
   S708_LM_DC_1ST_CLAMP1.Visu_Adv_Arr[2] := FALSE;
   S708_LM_DC_1ST_CLAMP1.Visu_Adv_Arr[3] := FALSE;
   S708_LM_DC_1ST_CLAMP1.Visu_Adv_Arr[4] := FALSE;
   S708_LM_DC_1ST_CLAMP1.Visu_Adv_Arr[5] := FALSE;
   S708_LM_DC_1ST_CLAMP1.Visu_Adv_Arr[6] := FALSE;
   S708_LM_DC_1ST_CLAMP1.Visu_Adv_Arr[7] := FALSE;
   S708_LM_DC_1ST_CLAMP1.Visu_Adv_Arr[8] := FALSE;
   S708_LM_DC_1ST_CLAMP1.Visu_Adv_Arr[9] := FALSE;
   S708_LM_DC_1ST_CLAMP1.Visu_Adv_Arr[10] := FALSE;
   S708_LM_DC_1ST_CLAMP1.Visu_Adv_Arr[11] := FALSE;
   S708_LM_DC_1ST_CLAMP1.Visu_Adv_Arr[12] := FALSE;
   S708_LM_DC_1ST_CLAMP1.Visu_Adv_Arr[13] := FALSE;
   S708_LM_DC_1ST_CLAMP1.Visu_Adv_Arr[14] := FALSE;
   S708_LM_DC_1ST_CLAMP1.Visu_Adv_Arr[15] := FALSE;
   S708_LM_DC_1ST_CLAMP1.Visu_Ret_Arr[0] := FALSE;
   S708_LM_DC_1ST_CLAMP1.Visu_Ret_Arr[1] := FALSE;
   S708_LM_DC_1ST_CLAMP1.Visu_Ret_Arr[2] := FALSE;
   S708_LM_DC_1ST_CLAMP1.Visu_Ret_Arr[3] := FALSE;
   S708_LM_DC_1ST_CLAMP1.Visu_Ret_Arr[4] := FALSE;
   S708_LM_DC_1ST_CLAMP1.Visu_Ret_Arr[5] := FALSE;
   S708_LM_DC_1ST_CLAMP1.Visu_Ret_Arr[6] := FALSE;
   S708_LM_DC_1ST_CLAMP1.Visu_Ret_Arr[7] := FALSE;
   S708_LM_DC_1ST_CLAMP1.Visu_Ret_Arr[8] := FALSE;
   S708_LM_DC_1ST_CLAMP1.Visu_Ret_Arr[9] := FALSE;
   S708_LM_DC_1ST_CLAMP1.Visu_Ret_Arr[10] := FALSE;
   S708_LM_DC_1ST_CLAMP1.Visu_Ret_Arr[11] := FALSE;
   S708_LM_DC_1ST_CLAMP1.Visu_Ret_Arr[12] := FALSE;
   S708_LM_DC_1ST_CLAMP1.Visu_Ret_Arr[13] := FALSE;
   S708_LM_DC_1ST_CLAMP1.Visu_Ret_Arr[14] := FALSE;
   S708_LM_DC_1ST_CLAMP1.Visu_Ret_Arr[15] := FALSE;
   S708_LM_DC_1ST_CLAMP1.BLK_Move_Ret := 0;
   S708_LM_DC_1ST_CLAMP1.Enable := FALSE;
   S708_LM_DC_1ST_CLAMP1.Adv_End := FALSE;
   S708_LM_DC_1ST_CLAMP1.Ret_End := FALSE;
   S708_LM_DC_1ST_CLAMP2.Enable_Aux := FALSE;
   S708_LM_DC_1ST_CLAMP2.Adv_Amount := 2;
   S708_LM_DC_1ST_CLAMP2.Ret_Amount := 2;
   S708_LM_DC_1ST_CLAMP2.LS_Adv1 := FALSE;
   S708_LM_DC_1ST_CLAMP2.LS_Ret1 := FALSE;
   S708_LM_DC_1ST_CLAMP2.LS_Adv2 := FALSE;
   S708_LM_DC_1ST_CLAMP2.LS_Ret2 := FALSE;
   S708_LM_DC_1ST_CLAMP2.LS_Adv3 := FALSE;
   S708_LM_DC_1ST_CLAMP2.LS_Ret3 := FALSE;
   S708_LM_DC_1ST_CLAMP2.LS_Adv4 := FALSE;
   S708_LM_DC_1ST_CLAMP2.LS_Ret4 := FALSE;
   S708_LM_DC_1ST_CLAMP2.SOL_Adv := FALSE;
   S708_LM_DC_1ST_CLAMP2.SOL_Ret := FALSE;
   S708_LM_DC_1ST_CLAMP2.M_Ready := TRUE;
   S708_LM_DC_1ST_CLAMP2.T_CHK1 := T#4S;
   S708_LM_DC_1ST_CLAMP2.T_CHK2 := T#4S;
   S708_LM_DC_1ST_CLAMP2.PB_Lamp_CHK := FALSE;
   S708_LM_DC_1ST_CLAMP2.PB_Error_Rst := FALSE;
   S708_LM_DC_1ST_CLAMP2.M_FLICK := FALSE;
   S708_LM_DC_1ST_CLAMP2.M_Adv_Err := FALSE;
   S708_LM_DC_1ST_CLAMP2.M_Ret_Err := FALSE;
   S708_LM_DC_1ST_CLAMP2.LP_Adv := FALSE;
   S708_LM_DC_1ST_CLAMP2.LP_Ret := FALSE;
   S708_LM_DC_1ST_CLAMP2.Visu_Adv := W#16#0;
   S708_LM_DC_1ST_CLAMP2.Visu_Ret := W#16#0;
   S708_LM_DC_1ST_CLAMP2.Error_T1.IN := FALSE;
   S708_LM_DC_1ST_CLAMP2.Error_T1.PT := T#4S;
   S708_LM_DC_1ST_CLAMP2.Error_T1.Q := FALSE;
   S708_LM_DC_1ST_CLAMP2.Error_T1.ET := T#0MS;
   S708_LM_DC_1ST_CLAMP2.Error_T1.STATE := B#16#0;
   S708_LM_DC_1ST_CLAMP2.Error_T1.STIME := T#22D23H1M3S514MS;
   S708_LM_DC_1ST_CLAMP2.Error_T1.ATIME := T#22D23H1M4S193MS;
   S708_LM_DC_1ST_CLAMP2.Error_T2.IN := FALSE;
   S708_LM_DC_1ST_CLAMP2.Error_T2.PT := T#4S;
   S708_LM_DC_1ST_CLAMP2.Error_T2.Q := FALSE;
   S708_LM_DC_1ST_CLAMP2.Error_T2.ET := T#0MS;
   S708_LM_DC_1ST_CLAMP2.Error_T2.STATE := B#16#0;
   S708_LM_DC_1ST_CLAMP2.Error_T2.STIME := T#0MS;
   S708_LM_DC_1ST_CLAMP2.Error_T2.ATIME := T#0MS;
   S708_LM_DC_1ST_CLAMP2.CHK_Aux1 := FALSE;
   S708_LM_DC_1ST_CLAMP2.CHK_Aux2 := FALSE;
   S708_LM_DC_1ST_CLAMP2.Error_T1_DN := FALSE;
   S708_LM_DC_1ST_CLAMP2.Error_T2_DN := FALSE;
   S708_LM_DC_1ST_CLAMP2.Adv_Memo := FALSE;
   S708_LM_DC_1ST_CLAMP2.Visu_Adv_Arr[0] := FALSE;
   S708_LM_DC_1ST_CLAMP2.Visu_Adv_Arr[1] := FALSE;
   S708_LM_DC_1ST_CLAMP2.Visu_Adv_Arr[2] := FALSE;
   S708_LM_DC_1ST_CLAMP2.Visu_Adv_Arr[3] := FALSE;
   S708_LM_DC_1ST_CLAMP2.Visu_Adv_Arr[4] := FALSE;
   S708_LM_DC_1ST_CLAMP2.Visu_Adv_Arr[5] := FALSE;
   S708_LM_DC_1ST_CLAMP2.Visu_Adv_Arr[6] := FALSE;
   S708_LM_DC_1ST_CLAMP2.Visu_Adv_Arr[7] := FALSE;
   S708_LM_DC_1ST_CLAMP2.Visu_Adv_Arr[8] := FALSE;
   S708_LM_DC_1ST_CLAMP2.Visu_Adv_Arr[9] := FALSE;
   S708_LM_DC_1ST_CLAMP2.Visu_Adv_Arr[10] := FALSE;
   S708_LM_DC_1ST_CLAMP2.Visu_Adv_Arr[11] := FALSE;
   S708_LM_DC_1ST_CLAMP2.Visu_Adv_Arr[12] := FALSE;
   S708_LM_DC_1ST_CLAMP2.Visu_Adv_Arr[13] := FALSE;
   S708_LM_DC_1ST_CLAMP2.Visu_Adv_Arr[14] := FALSE;
   S708_LM_DC_1ST_CLAMP2.Visu_Adv_Arr[15] := FALSE;
   S708_LM_DC_1ST_CLAMP2.Visu_Ret_Arr[0] := FALSE;
   S708_LM_DC_1ST_CLAMP2.Visu_Ret_Arr[1] := FALSE;
   S708_LM_DC_1ST_CLAMP2.Visu_Ret_Arr[2] := FALSE;
   S708_LM_DC_1ST_CLAMP2.Visu_Ret_Arr[3] := FALSE;
   S708_LM_DC_1ST_CLAMP2.Visu_Ret_Arr[4] := FALSE;
   S708_LM_DC_1ST_CLAMP2.Visu_Ret_Arr[5] := FALSE;
   S708_LM_DC_1ST_CLAMP2.Visu_Ret_Arr[6] := FALSE;
   S708_LM_DC_1ST_CLAMP2.Visu_Ret_Arr[7] := FALSE;
   S708_LM_DC_1ST_CLAMP2.Visu_Ret_Arr[8] := FALSE;
   S708_LM_DC_1ST_CLAMP2.Visu_Ret_Arr[9] := FALSE;
   S708_LM_DC_1ST_CLAMP2.Visu_Ret_Arr[10] := FALSE;
   S708_LM_DC_1ST_CLAMP2.Visu_Ret_Arr[11] := FALSE;
   S708_LM_DC_1ST_CLAMP2.Visu_Ret_Arr[12] := FALSE;
   S708_LM_DC_1ST_CLAMP2.Visu_Ret_Arr[13] := FALSE;
   S708_LM_DC_1ST_CLAMP2.Visu_Ret_Arr[14] := FALSE;
   S708_LM_DC_1ST_CLAMP2.Visu_Ret_Arr[15] := FALSE;
   S708_LM_DC_1ST_CLAMP2.BLK_Move_Ret := 0;
   S708_LM_DC_1ST_CLAMP2.Enable := FALSE;
   S708_LM_DC_1ST_CLAMP2.Adv_End := FALSE;
   S708_LM_DC_1ST_CLAMP2.Ret_End := FALSE;
   S708_LM_DC_1ST_CLAMP3.Enable_Aux := FALSE;
   S708_LM_DC_1ST_CLAMP3.Adv_Amount := 1;
   S708_LM_DC_1ST_CLAMP3.Ret_Amount := 1;
   S708_LM_DC_1ST_CLAMP3.LS_Adv1 := FALSE;
   S708_LM_DC_1ST_CLAMP3.LS_Ret1 := FALSE;
   S708_LM_DC_1ST_CLAMP3.LS_Adv2 := FALSE;
   S708_LM_DC_1ST_CLAMP3.LS_Ret2 := FALSE;
   S708_LM_DC_1ST_CLAMP3.LS_Adv3 := FALSE;
   S708_LM_DC_1ST_CLAMP3.LS_Ret3 := FALSE;
   S708_LM_DC_1ST_CLAMP3.LS_Adv4 := FALSE;
   S708_LM_DC_1ST_CLAMP3.LS_Ret4 := FALSE;
   S708_LM_DC_1ST_CLAMP3.SOL_Adv := FALSE;
   S708_LM_DC_1ST_CLAMP3.SOL_Ret := FALSE;
   S708_LM_DC_1ST_CLAMP3.M_Ready := TRUE;
   S708_LM_DC_1ST_CLAMP3.T_CHK1 := T#4S;
   S708_LM_DC_1ST_CLAMP3.T_CHK2 := T#4S;
   S708_LM_DC_1ST_CLAMP3.PB_Lamp_CHK := FALSE;
   S708_LM_DC_1ST_CLAMP3.PB_Error_Rst := FALSE;
   S708_LM_DC_1ST_CLAMP3.M_FLICK := FALSE;
   S708_LM_DC_1ST_CLAMP3.M_Adv_Err := FALSE;
   S708_LM_DC_1ST_CLAMP3.M_Ret_Err := FALSE;
   S708_LM_DC_1ST_CLAMP3.LP_Adv := FALSE;
   S708_LM_DC_1ST_CLAMP3.LP_Ret := FALSE;
   S708_LM_DC_1ST_CLAMP3.Visu_Adv := W#16#0;
   S708_LM_DC_1ST_CLAMP3.Visu_Ret := W#16#0;
   S708_LM_DC_1ST_CLAMP3.Error_T1.IN := FALSE;
   S708_LM_DC_1ST_CLAMP3.Error_T1.PT := T#4S;
   S708_LM_DC_1ST_CLAMP3.Error_T1.Q := FALSE;
   S708_LM_DC_1ST_CLAMP3.Error_T1.ET := T#0MS;
   S708_LM_DC_1ST_CLAMP3.Error_T1.STATE := B#16#0;
   S708_LM_DC_1ST_CLAMP3.Error_T1.STIME := T#0MS;
   S708_LM_DC_1ST_CLAMP3.Error_T1.ATIME := T#0MS;
   S708_LM_DC_1ST_CLAMP3.Error_T2.IN := FALSE;
   S708_LM_DC_1ST_CLAMP3.Error_T2.PT := T#4S;
   S708_LM_DC_1ST_CLAMP3.Error_T2.Q := FALSE;
   S708_LM_DC_1ST_CLAMP3.Error_T2.ET := T#0MS;
   S708_LM_DC_1ST_CLAMP3.Error_T2.STATE := B#16#0;
   S708_LM_DC_1ST_CLAMP3.Error_T2.STIME := T#0MS;
   S708_LM_DC_1ST_CLAMP3.Error_T2.ATIME := T#0MS;
   S708_LM_DC_1ST_CLAMP3.CHK_Aux1 := FALSE;
   S708_LM_DC_1ST_CLAMP3.CHK_Aux2 := FALSE;
   S708_LM_DC_1ST_CLAMP3.Error_T1_DN := FALSE;
   S708_LM_DC_1ST_CLAMP3.Error_T2_DN := FALSE;
   S708_LM_DC_1ST_CLAMP3.Adv_Memo := FALSE;
   S708_LM_DC_1ST_CLAMP3.Visu_Adv_Arr[0] := FALSE;
   S708_LM_DC_1ST_CLAMP3.Visu_Adv_Arr[1] := FALSE;
   S708_LM_DC_1ST_CLAMP3.Visu_Adv_Arr[2] := FALSE;
   S708_LM_DC_1ST_CLAMP3.Visu_Adv_Arr[3] := FALSE;
   S708_LM_DC_1ST_CLAMP3.Visu_Adv_Arr[4] := FALSE;
   S708_LM_DC_1ST_CLAMP3.Visu_Adv_Arr[5] := FALSE;
   S708_LM_DC_1ST_CLAMP3.Visu_Adv_Arr[6] := FALSE;
   S708_LM_DC_1ST_CLAMP3.Visu_Adv_Arr[7] := FALSE;
   S708_LM_DC_1ST_CLAMP3.Visu_Adv_Arr[8] := FALSE;
   S708_LM_DC_1ST_CLAMP3.Visu_Adv_Arr[9] := FALSE;
   S708_LM_DC_1ST_CLAMP3.Visu_Adv_Arr[10] := FALSE;
   S708_LM_DC_1ST_CLAMP3.Visu_Adv_Arr[11] := FALSE;
   S708_LM_DC_1ST_CLAMP3.Visu_Adv_Arr[12] := FALSE;
   S708_LM_DC_1ST_CLAMP3.Visu_Adv_Arr[13] := FALSE;
   S708_LM_DC_1ST_CLAMP3.Visu_Adv_Arr[14] := FALSE;
   S708_LM_DC_1ST_CLAMP3.Visu_Adv_Arr[15] := FALSE;
   S708_LM_DC_1ST_CLAMP3.Visu_Ret_Arr[0] := FALSE;
   S708_LM_DC_1ST_CLAMP3.Visu_Ret_Arr[1] := FALSE;
   S708_LM_DC_1ST_CLAMP3.Visu_Ret_Arr[2] := FALSE;
   S708_LM_DC_1ST_CLAMP3.Visu_Ret_Arr[3] := FALSE;
   S708_LM_DC_1ST_CLAMP3.Visu_Ret_Arr[4] := FALSE;
   S708_LM_DC_1ST_CLAMP3.Visu_Ret_Arr[5] := FALSE;
   S708_LM_DC_1ST_CLAMP3.Visu_Ret_Arr[6] := FALSE;
   S708_LM_DC_1ST_CLAMP3.Visu_Ret_Arr[7] := FALSE;
   S708_LM_DC_1ST_CLAMP3.Visu_Ret_Arr[8] := FALSE;
   S708_LM_DC_1ST_CLAMP3.Visu_Ret_Arr[9] := FALSE;
   S708_LM_DC_1ST_CLAMP3.Visu_Ret_Arr[10] := FALSE;
   S708_LM_DC_1ST_CLAMP3.Visu_Ret_Arr[11] := FALSE;
   S708_LM_DC_1ST_CLAMP3.Visu_Ret_Arr[12] := FALSE;
   S708_LM_DC_1ST_CLAMP3.Visu_Ret_Arr[13] := FALSE;
   S708_LM_DC_1ST_CLAMP3.Visu_Ret_Arr[14] := FALSE;
   S708_LM_DC_1ST_CLAMP3.Visu_Ret_Arr[15] := FALSE;
   S708_LM_DC_1ST_CLAMP3.BLK_Move_Ret := 0;
   S708_LM_DC_1ST_CLAMP3.Enable := FALSE;
   S708_LM_DC_1ST_CLAMP3.Adv_End := FALSE;
   S708_LM_DC_1ST_CLAMP3.Ret_End := FALSE;
   S708_LM_DC_1ST_CLAMP4.Enable_Aux := FALSE;
   S708_LM_DC_1ST_CLAMP4.Adv_Amount := 1;
   S708_LM_DC_1ST_CLAMP4.Ret_Amount := 1;
   S708_LM_DC_1ST_CLAMP4.LS_Adv1 := FALSE;
   S708_LM_DC_1ST_CLAMP4.LS_Ret1 := FALSE;
   S708_LM_DC_1ST_CLAMP4.LS_Adv2 := FALSE;
   S708_LM_DC_1ST_CLAMP4.LS_Ret2 := FALSE;
   S708_LM_DC_1ST_CLAMP4.LS_Adv3 := FALSE;
   S708_LM_DC_1ST_CLAMP4.LS_Ret3 := FALSE;
   S708_LM_DC_1ST_CLAMP4.LS_Adv4 := FALSE;
   S708_LM_DC_1ST_CLAMP4.LS_Ret4 := FALSE;
   S708_LM_DC_1ST_CLAMP4.SOL_Adv := FALSE;
   S708_LM_DC_1ST_CLAMP4.SOL_Ret := FALSE;
   S708_LM_DC_1ST_CLAMP4.M_Ready := TRUE;
   S708_LM_DC_1ST_CLAMP4.T_CHK1 := T#4S;
   S708_LM_DC_1ST_CLAMP4.T_CHK2 := T#4S;
   S708_LM_DC_1ST_CLAMP4.PB_Lamp_CHK := FALSE;
   S708_LM_DC_1ST_CLAMP4.PB_Error_Rst := FALSE;
   S708_LM_DC_1ST_CLAMP4.M_FLICK := FALSE;
   S708_LM_DC_1ST_CLAMP4.M_Adv_Err := FALSE;
   S708_LM_DC_1ST_CLAMP4.M_Ret_Err := FALSE;
   S708_LM_DC_1ST_CLAMP4.LP_Adv := FALSE;
   S708_LM_DC_1ST_CLAMP4.LP_Ret := FALSE;
   S708_LM_DC_1ST_CLAMP4.Visu_Adv := W#16#0;
   S708_LM_DC_1ST_CLAMP4.Visu_Ret := W#16#0;
   S708_LM_DC_1ST_CLAMP4.Error_T1.IN := FALSE;
   S708_LM_DC_1ST_CLAMP4.Error_T1.PT := T#4S;
   S708_LM_DC_1ST_CLAMP4.Error_T1.Q := FALSE;
   S708_LM_DC_1ST_CLAMP4.Error_T1.ET := T#0MS;
   S708_LM_DC_1ST_CLAMP4.Error_T1.STATE := B#16#0;
   S708_LM_DC_1ST_CLAMP4.Error_T1.STIME := T#0MS;
   S708_LM_DC_1ST_CLAMP4.Error_T1.ATIME := T#0MS;
   S708_LM_DC_1ST_CLAMP4.Error_T2.IN := FALSE;
   S708_LM_DC_1ST_CLAMP4.Error_T2.PT := T#4S;
   S708_LM_DC_1ST_CLAMP4.Error_T2.Q := FALSE;
   S708_LM_DC_1ST_CLAMP4.Error_T2.ET := T#0MS;
   S708_LM_DC_1ST_CLAMP4.Error_T2.STATE := B#16#0;
   S708_LM_DC_1ST_CLAMP4.Error_T2.STIME := T#0MS;
   S708_LM_DC_1ST_CLAMP4.Error_T2.ATIME := T#0MS;
   S708_LM_DC_1ST_CLAMP4.CHK_Aux1 := FALSE;
   S708_LM_DC_1ST_CLAMP4.CHK_Aux2 := FALSE;
   S708_LM_DC_1ST_CLAMP4.Error_T1_DN := FALSE;
   S708_LM_DC_1ST_CLAMP4.Error_T2_DN := FALSE;
   S708_LM_DC_1ST_CLAMP4.Adv_Memo := FALSE;
   S708_LM_DC_1ST_CLAMP4.Visu_Adv_Arr[0] := FALSE;
   S708_LM_DC_1ST_CLAMP4.Visu_Adv_Arr[1] := FALSE;
   S708_LM_DC_1ST_CLAMP4.Visu_Adv_Arr[2] := FALSE;
   S708_LM_DC_1ST_CLAMP4.Visu_Adv_Arr[3] := FALSE;
   S708_LM_DC_1ST_CLAMP4.Visu_Adv_Arr[4] := FALSE;
   S708_LM_DC_1ST_CLAMP4.Visu_Adv_Arr[5] := FALSE;
   S708_LM_DC_1ST_CLAMP4.Visu_Adv_Arr[6] := FALSE;
   S708_LM_DC_1ST_CLAMP4.Visu_Adv_Arr[7] := FALSE;
   S708_LM_DC_1ST_CLAMP4.Visu_Adv_Arr[8] := FALSE;
   S708_LM_DC_1ST_CLAMP4.Visu_Adv_Arr[9] := FALSE;
   S708_LM_DC_1ST_CLAMP4.Visu_Adv_Arr[10] := FALSE;
   S708_LM_DC_1ST_CLAMP4.Visu_Adv_Arr[11] := FALSE;
   S708_LM_DC_1ST_CLAMP4.Visu_Adv_Arr[12] := FALSE;
   S708_LM_DC_1ST_CLAMP4.Visu_Adv_Arr[13] := FALSE;
   S708_LM_DC_1ST_CLAMP4.Visu_Adv_Arr[14] := FALSE;
   S708_LM_DC_1ST_CLAMP4.Visu_Adv_Arr[15] := FALSE;
   S708_LM_DC_1ST_CLAMP4.Visu_Ret_Arr[0] := FALSE;
   S708_LM_DC_1ST_CLAMP4.Visu_Ret_Arr[1] := FALSE;
   S708_LM_DC_1ST_CLAMP4.Visu_Ret_Arr[2] := FALSE;
   S708_LM_DC_1ST_CLAMP4.Visu_Ret_Arr[3] := FALSE;
   S708_LM_DC_1ST_CLAMP4.Visu_Ret_Arr[4] := FALSE;
   S708_LM_DC_1ST_CLAMP4.Visu_Ret_Arr[5] := FALSE;
   S708_LM_DC_1ST_CLAMP4.Visu_Ret_Arr[6] := FALSE;
   S708_LM_DC_1ST_CLAMP4.Visu_Ret_Arr[7] := FALSE;
   S708_LM_DC_1ST_CLAMP4.Visu_Ret_Arr[8] := FALSE;
   S708_LM_DC_1ST_CLAMP4.Visu_Ret_Arr[9] := FALSE;
   S708_LM_DC_1ST_CLAMP4.Visu_Ret_Arr[10] := FALSE;
   S708_LM_DC_1ST_CLAMP4.Visu_Ret_Arr[11] := FALSE;
   S708_LM_DC_1ST_CLAMP4.Visu_Ret_Arr[12] := FALSE;
   S708_LM_DC_1ST_CLAMP4.Visu_Ret_Arr[13] := FALSE;
   S708_LM_DC_1ST_CLAMP4.Visu_Ret_Arr[14] := FALSE;
   S708_LM_DC_1ST_CLAMP4.Visu_Ret_Arr[15] := FALSE;
   S708_LM_DC_1ST_CLAMP4.BLK_Move_Ret := 0;
   S708_LM_DC_1ST_CLAMP4.Enable := FALSE;
   S708_LM_DC_1ST_CLAMP4.Adv_End := FALSE;
   S708_LM_DC_1ST_CLAMP4.Ret_End := FALSE;
   S708_LM_DC_2ND_CLAMP1.Enable_Aux := FALSE;
   S708_LM_DC_2ND_CLAMP1.Adv_Amount := 1;
   S708_LM_DC_2ND_CLAMP1.Ret_Amount := 1;
   S708_LM_DC_2ND_CLAMP1.LS_Adv1 := FALSE;
   S708_LM_DC_2ND_CLAMP1.LS_Ret1 := FALSE;
   S708_LM_DC_2ND_CLAMP1.LS_Adv2 := FALSE;
   S708_LM_DC_2ND_CLAMP1.LS_Ret2 := FALSE;
   S708_LM_DC_2ND_CLAMP1.LS_Adv3 := FALSE;
   S708_LM_DC_2ND_CLAMP1.LS_Ret3 := FALSE;
   S708_LM_DC_2ND_CLAMP1.LS_Adv4 := FALSE;
   S708_LM_DC_2ND_CLAMP1.LS_Ret4 := FALSE;
   S708_LM_DC_2ND_CLAMP1.SOL_Adv := FALSE;
   S708_LM_DC_2ND_CLAMP1.SOL_Ret := FALSE;
   S708_LM_DC_2ND_CLAMP1.M_Ready := TRUE;
   S708_LM_DC_2ND_CLAMP1.T_CHK1 := T#4S;
   S708_LM_DC_2ND_CLAMP1.T_CHK2 := T#4S;
   S708_LM_DC_2ND_CLAMP1.PB_Lamp_CHK := FALSE;
   S708_LM_DC_2ND_CLAMP1.PB_Error_Rst := FALSE;
   S708_LM_DC_2ND_CLAMP1.M_FLICK := FALSE;
   S708_LM_DC_2ND_CLAMP1.M_Adv_Err := FALSE;
   S708_LM_DC_2ND_CLAMP1.M_Ret_Err := FALSE;
   S708_LM_DC_2ND_CLAMP1.LP_Adv := FALSE;
   S708_LM_DC_2ND_CLAMP1.LP_Ret := FALSE;
   S708_LM_DC_2ND_CLAMP1.Visu_Adv := W#16#0;
   S708_LM_DC_2ND_CLAMP1.Visu_Ret := W#16#0;
   S708_LM_DC_2ND_CLAMP1.Error_T1.IN := FALSE;
   S708_LM_DC_2ND_CLAMP1.Error_T1.PT := T#4S;
   S708_LM_DC_2ND_CLAMP1.Error_T1.Q := FALSE;
   S708_LM_DC_2ND_CLAMP1.Error_T1.ET := T#0MS;
   S708_LM_DC_2ND_CLAMP1.Error_T1.STATE := B#16#0;
   S708_LM_DC_2ND_CLAMP1.Error_T1.STIME := T#22D23H1M2S540MS;
   S708_LM_DC_2ND_CLAMP1.Error_T1.ATIME := T#22D23H1M4S149MS;
   S708_LM_DC_2ND_CLAMP1.Error_T2.IN := FALSE;
   S708_LM_DC_2ND_CLAMP1.Error_T2.PT := T#4S;
   S708_LM_DC_2ND_CLAMP1.Error_T2.Q := FALSE;
   S708_LM_DC_2ND_CLAMP1.Error_T2.ET := T#0MS;
   S708_LM_DC_2ND_CLAMP1.Error_T2.STATE := B#16#0;
   S708_LM_DC_2ND_CLAMP1.Error_T2.STIME := T#0MS;
   S708_LM_DC_2ND_CLAMP1.Error_T2.ATIME := T#0MS;
   S708_LM_DC_2ND_CLAMP1.CHK_Aux1 := FALSE;
   S708_LM_DC_2ND_CLAMP1.CHK_Aux2 := FALSE;
   S708_LM_DC_2ND_CLAMP1.Error_T1_DN := FALSE;
   S708_LM_DC_2ND_CLAMP1.Error_T2_DN := FALSE;
   S708_LM_DC_2ND_CLAMP1.Adv_Memo := FALSE;
   S708_LM_DC_2ND_CLAMP1.Visu_Adv_Arr[0] := FALSE;
   S708_LM_DC_2ND_CLAMP1.Visu_Adv_Arr[1] := FALSE;
   S708_LM_DC_2ND_CLAMP1.Visu_Adv_Arr[2] := FALSE;
   S708_LM_DC_2ND_CLAMP1.Visu_Adv_Arr[3] := FALSE;
   S708_LM_DC_2ND_CLAMP1.Visu_Adv_Arr[4] := FALSE;
   S708_LM_DC_2ND_CLAMP1.Visu_Adv_Arr[5] := FALSE;
   S708_LM_DC_2ND_CLAMP1.Visu_Adv_Arr[6] := FALSE;
   S708_LM_DC_2ND_CLAMP1.Visu_Adv_Arr[7] := FALSE;
   S708_LM_DC_2ND_CLAMP1.Visu_Adv_Arr[8] := FALSE;
   S708_LM_DC_2ND_CLAMP1.Visu_Adv_Arr[9] := FALSE;
   S708_LM_DC_2ND_CLAMP1.Visu_Adv_Arr[10] := FALSE;
   S708_LM_DC_2ND_CLAMP1.Visu_Adv_Arr[11] := FALSE;
   S708_LM_DC_2ND_CLAMP1.Visu_Adv_Arr[12] := FALSE;
   S708_LM_DC_2ND_CLAMP1.Visu_Adv_Arr[13] := FALSE;
   S708_LM_DC_2ND_CLAMP1.Visu_Adv_Arr[14] := FALSE;
   S708_LM_DC_2ND_CLAMP1.Visu_Adv_Arr[15] := FALSE;
   S708_LM_DC_2ND_CLAMP1.Visu_Ret_Arr[0] := FALSE;
   S708_LM_DC_2ND_CLAMP1.Visu_Ret_Arr[1] := FALSE;
   S708_LM_DC_2ND_CLAMP1.Visu_Ret_Arr[2] := FALSE;
   S708_LM_DC_2ND_CLAMP1.Visu_Ret_Arr[3] := FALSE;
   S708_LM_DC_2ND_CLAMP1.Visu_Ret_Arr[4] := FALSE;
   S708_LM_DC_2ND_CLAMP1.Visu_Ret_Arr[5] := FALSE;
   S708_LM_DC_2ND_CLAMP1.Visu_Ret_Arr[6] := FALSE;
   S708_LM_DC_2ND_CLAMP1.Visu_Ret_Arr[7] := FALSE;
   S708_LM_DC_2ND_CLAMP1.Visu_Ret_Arr[8] := FALSE;
   S708_LM_DC_2ND_CLAMP1.Visu_Ret_Arr[9] := FALSE;
   S708_LM_DC_2ND_CLAMP1.Visu_Ret_Arr[10] := FALSE;
   S708_LM_DC_2ND_CLAMP1.Visu_Ret_Arr[11] := FALSE;
   S708_LM_DC_2ND_CLAMP1.Visu_Ret_Arr[12] := FALSE;
   S708_LM_DC_2ND_CLAMP1.Visu_Ret_Arr[13] := FALSE;
   S708_LM_DC_2ND_CLAMP1.Visu_Ret_Arr[14] := FALSE;
   S708_LM_DC_2ND_CLAMP1.Visu_Ret_Arr[15] := FALSE;
   S708_LM_DC_2ND_CLAMP1.BLK_Move_Ret := 0;
   S708_LM_DC_2ND_CLAMP1.Enable := FALSE;
   S708_LM_DC_2ND_CLAMP1.Adv_End := FALSE;
   S708_LM_DC_2ND_CLAMP1.Ret_End := FALSE;
   S708_LM_DC_2ND_CLAMP2.Enable_Aux := FALSE;
   S708_LM_DC_2ND_CLAMP2.Adv_Amount := 1;
   S708_LM_DC_2ND_CLAMP2.Ret_Amount := 1;
   S708_LM_DC_2ND_CLAMP2.LS_Adv1 := FALSE;
   S708_LM_DC_2ND_CLAMP2.LS_Ret1 := FALSE;
   S708_LM_DC_2ND_CLAMP2.LS_Adv2 := FALSE;
   S708_LM_DC_2ND_CLAMP2.LS_Ret2 := FALSE;
   S708_LM_DC_2ND_CLAMP2.LS_Adv3 := FALSE;
   S708_LM_DC_2ND_CLAMP2.LS_Ret3 := FALSE;
   S708_LM_DC_2ND_CLAMP2.LS_Adv4 := FALSE;
   S708_LM_DC_2ND_CLAMP2.LS_Ret4 := FALSE;
   S708_LM_DC_2ND_CLAMP2.SOL_Adv := FALSE;
   S708_LM_DC_2ND_CLAMP2.SOL_Ret := FALSE;
   S708_LM_DC_2ND_CLAMP2.M_Ready := TRUE;
   S708_LM_DC_2ND_CLAMP2.T_CHK1 := T#4S;
   S708_LM_DC_2ND_CLAMP2.T_CHK2 := T#4S;
   S708_LM_DC_2ND_CLAMP2.PB_Lamp_CHK := FALSE;
   S708_LM_DC_2ND_CLAMP2.PB_Error_Rst := FALSE;
   S708_LM_DC_2ND_CLAMP2.M_FLICK := FALSE;
   S708_LM_DC_2ND_CLAMP2.M_Adv_Err := FALSE;
   S708_LM_DC_2ND_CLAMP2.M_Ret_Err := FALSE;
   S708_LM_DC_2ND_CLAMP2.LP_Adv := FALSE;
   S708_LM_DC_2ND_CLAMP2.LP_Ret := FALSE;
   S708_LM_DC_2ND_CLAMP2.Visu_Adv := W#16#0;
   S708_LM_DC_2ND_CLAMP2.Visu_Ret := W#16#0;
   S708_LM_DC_2ND_CLAMP2.Error_T1.IN := FALSE;
   S708_LM_DC_2ND_CLAMP2.Error_T1.PT := T#4S;
   S708_LM_DC_2ND_CLAMP2.Error_T1.Q := FALSE;
   S708_LM_DC_2ND_CLAMP2.Error_T1.ET := T#0MS;
   S708_LM_DC_2ND_CLAMP2.Error_T1.STATE := B#16#0;
   S708_LM_DC_2ND_CLAMP2.Error_T1.STIME := T#22D23H1M2S540MS;
   S708_LM_DC_2ND_CLAMP2.Error_T1.ATIME := T#22D23H1M4S238MS;
   S708_LM_DC_2ND_CLAMP2.Error_T2.IN := FALSE;
   S708_LM_DC_2ND_CLAMP2.Error_T2.PT := T#4S;
   S708_LM_DC_2ND_CLAMP2.Error_T2.Q := FALSE;
   S708_LM_DC_2ND_CLAMP2.Error_T2.ET := T#0MS;
   S708_LM_DC_2ND_CLAMP2.Error_T2.STATE := B#16#0;
   S708_LM_DC_2ND_CLAMP2.Error_T2.STIME := T#0MS;
   S708_LM_DC_2ND_CLAMP2.Error_T2.ATIME := T#0MS;
   S708_LM_DC_2ND_CLAMP2.CHK_Aux1 := FALSE;
   S708_LM_DC_2ND_CLAMP2.CHK_Aux2 := FALSE;
   S708_LM_DC_2ND_CLAMP2.Error_T1_DN := FALSE;
   S708_LM_DC_2ND_CLAMP2.Error_T2_DN := FALSE;
   S708_LM_DC_2ND_CLAMP2.Adv_Memo := FALSE;
   S708_LM_DC_2ND_CLAMP2.Visu_Adv_Arr[0] := FALSE;
   S708_LM_DC_2ND_CLAMP2.Visu_Adv_Arr[1] := FALSE;
   S708_LM_DC_2ND_CLAMP2.Visu_Adv_Arr[2] := FALSE;
   S708_LM_DC_2ND_CLAMP2.Visu_Adv_Arr[3] := FALSE;
   S708_LM_DC_2ND_CLAMP2.Visu_Adv_Arr[4] := FALSE;
   S708_LM_DC_2ND_CLAMP2.Visu_Adv_Arr[5] := FALSE;
   S708_LM_DC_2ND_CLAMP2.Visu_Adv_Arr[6] := FALSE;
   S708_LM_DC_2ND_CLAMP2.Visu_Adv_Arr[7] := FALSE;
   S708_LM_DC_2ND_CLAMP2.Visu_Adv_Arr[8] := FALSE;
   S708_LM_DC_2ND_CLAMP2.Visu_Adv_Arr[9] := FALSE;
   S708_LM_DC_2ND_CLAMP2.Visu_Adv_Arr[10] := FALSE;
   S708_LM_DC_2ND_CLAMP2.Visu_Adv_Arr[11] := FALSE;
   S708_LM_DC_2ND_CLAMP2.Visu_Adv_Arr[12] := FALSE;
   S708_LM_DC_2ND_CLAMP2.Visu_Adv_Arr[13] := FALSE;
   S708_LM_DC_2ND_CLAMP2.Visu_Adv_Arr[14] := FALSE;
   S708_LM_DC_2ND_CLAMP2.Visu_Adv_Arr[15] := FALSE;
   S708_LM_DC_2ND_CLAMP2.Visu_Ret_Arr[0] := FALSE;
   S708_LM_DC_2ND_CLAMP2.Visu_Ret_Arr[1] := FALSE;
   S708_LM_DC_2ND_CLAMP2.Visu_Ret_Arr[2] := FALSE;
   S708_LM_DC_2ND_CLAMP2.Visu_Ret_Arr[3] := FALSE;
   S708_LM_DC_2ND_CLAMP2.Visu_Ret_Arr[4] := FALSE;
   S708_LM_DC_2ND_CLAMP2.Visu_Ret_Arr[5] := FALSE;
   S708_LM_DC_2ND_CLAMP2.Visu_Ret_Arr[6] := FALSE;
   S708_LM_DC_2ND_CLAMP2.Visu_Ret_Arr[7] := FALSE;
   S708_LM_DC_2ND_CLAMP2.Visu_Ret_Arr[8] := FALSE;
   S708_LM_DC_2ND_CLAMP2.Visu_Ret_Arr[9] := FALSE;
   S708_LM_DC_2ND_CLAMP2.Visu_Ret_Arr[10] := FALSE;
   S708_LM_DC_2ND_CLAMP2.Visu_Ret_Arr[11] := FALSE;
   S708_LM_DC_2ND_CLAMP2.Visu_Ret_Arr[12] := FALSE;
   S708_LM_DC_2ND_CLAMP2.Visu_Ret_Arr[13] := FALSE;
   S708_LM_DC_2ND_CLAMP2.Visu_Ret_Arr[14] := FALSE;
   S708_LM_DC_2ND_CLAMP2.Visu_Ret_Arr[15] := FALSE;
   S708_LM_DC_2ND_CLAMP2.BLK_Move_Ret := 0;
   S708_LM_DC_2ND_CLAMP2.Enable := FALSE;
   S708_LM_DC_2ND_CLAMP2.Adv_End := FALSE;
   S708_LM_DC_2ND_CLAMP2.Ret_End := FALSE;
   S708_LM_DC_2ND_CLAMP3.Enable_Aux := FALSE;
   S708_LM_DC_2ND_CLAMP3.Adv_Amount := 1;
   S708_LM_DC_2ND_CLAMP3.Ret_Amount := 1;
   S708_LM_DC_2ND_CLAMP3.LS_Adv1 := FALSE;
   S708_LM_DC_2ND_CLAMP3.LS_Ret1 := FALSE;
   S708_LM_DC_2ND_CLAMP3.LS_Adv2 := FALSE;
   S708_LM_DC_2ND_CLAMP3.LS_Ret2 := FALSE;
   S708_LM_DC_2ND_CLAMP3.LS_Adv3 := FALSE;
   S708_LM_DC_2ND_CLAMP3.LS_Ret3 := FALSE;
   S708_LM_DC_2ND_CLAMP3.LS_Adv4 := FALSE;
   S708_LM_DC_2ND_CLAMP3.LS_Ret4 := FALSE;
   S708_LM_DC_2ND_CLAMP3.SOL_Adv := FALSE;
   S708_LM_DC_2ND_CLAMP3.SOL_Ret := FALSE;
   S708_LM_DC_2ND_CLAMP3.M_Ready := TRUE;
   S708_LM_DC_2ND_CLAMP3.T_CHK1 := T#4S;
   S708_LM_DC_2ND_CLAMP3.T_CHK2 := T#4S;
   S708_LM_DC_2ND_CLAMP3.PB_Lamp_CHK := FALSE;
   S708_LM_DC_2ND_CLAMP3.PB_Error_Rst := FALSE;
   S708_LM_DC_2ND_CLAMP3.M_FLICK := FALSE;
   S708_LM_DC_2ND_CLAMP3.M_Adv_Err := FALSE;
   S708_LM_DC_2ND_CLAMP3.M_Ret_Err := FALSE;
   S708_LM_DC_2ND_CLAMP3.LP_Adv := FALSE;
   S708_LM_DC_2ND_CLAMP3.LP_Ret := FALSE;
   S708_LM_DC_2ND_CLAMP3.Visu_Adv := W#16#0;
   S708_LM_DC_2ND_CLAMP3.Visu_Ret := W#16#0;
   S708_LM_DC_2ND_CLAMP3.Error_T1.IN := FALSE;
   S708_LM_DC_2ND_CLAMP3.Error_T1.PT := T#4S;
   S708_LM_DC_2ND_CLAMP3.Error_T1.Q := FALSE;
   S708_LM_DC_2ND_CLAMP3.Error_T1.ET := T#0MS;
   S708_LM_DC_2ND_CLAMP3.Error_T1.STATE := B#16#0;
   S708_LM_DC_2ND_CLAMP3.Error_T1.STIME := T#22D23H1M2S540MS;
   S708_LM_DC_2ND_CLAMP3.Error_T1.ATIME := T#22D23H1M3S333MS;
   S708_LM_DC_2ND_CLAMP3.Error_T2.IN := FALSE;
   S708_LM_DC_2ND_CLAMP3.Error_T2.PT := T#4S;
   S708_LM_DC_2ND_CLAMP3.Error_T2.Q := FALSE;
   S708_LM_DC_2ND_CLAMP3.Error_T2.ET := T#0MS;
   S708_LM_DC_2ND_CLAMP3.Error_T2.STATE := B#16#0;
   S708_LM_DC_2ND_CLAMP3.Error_T2.STIME := T#0MS;
   S708_LM_DC_2ND_CLAMP3.Error_T2.ATIME := T#0MS;
   S708_LM_DC_2ND_CLAMP3.CHK_Aux1 := FALSE;
   S708_LM_DC_2ND_CLAMP3.CHK_Aux2 := FALSE;
   S708_LM_DC_2ND_CLAMP3.Error_T1_DN := FALSE;
   S708_LM_DC_2ND_CLAMP3.Error_T2_DN := FALSE;
   S708_LM_DC_2ND_CLAMP3.Adv_Memo := FALSE;
   S708_LM_DC_2ND_CLAMP3.Visu_Adv_Arr[0] := FALSE;
   S708_LM_DC_2ND_CLAMP3.Visu_Adv_Arr[1] := FALSE;
   S708_LM_DC_2ND_CLAMP3.Visu_Adv_Arr[2] := FALSE;
   S708_LM_DC_2ND_CLAMP3.Visu_Adv_Arr[3] := FALSE;
   S708_LM_DC_2ND_CLAMP3.Visu_Adv_Arr[4] := FALSE;
   S708_LM_DC_2ND_CLAMP3.Visu_Adv_Arr[5] := FALSE;
   S708_LM_DC_2ND_CLAMP3.Visu_Adv_Arr[6] := FALSE;
   S708_LM_DC_2ND_CLAMP3.Visu_Adv_Arr[7] := FALSE;
   S708_LM_DC_2ND_CLAMP3.Visu_Adv_Arr[8] := FALSE;
   S708_LM_DC_2ND_CLAMP3.Visu_Adv_Arr[9] := FALSE;
   S708_LM_DC_2ND_CLAMP3.Visu_Adv_Arr[10] := FALSE;
   S708_LM_DC_2ND_CLAMP3.Visu_Adv_Arr[11] := FALSE;
   S708_LM_DC_2ND_CLAMP3.Visu_Adv_Arr[12] := FALSE;
   S708_LM_DC_2ND_CLAMP3.Visu_Adv_Arr[13] := FALSE;
   S708_LM_DC_2ND_CLAMP3.Visu_Adv_Arr[14] := FALSE;
   S708_LM_DC_2ND_CLAMP3.Visu_Adv_Arr[15] := FALSE;
   S708_LM_DC_2ND_CLAMP3.Visu_Ret_Arr[0] := FALSE;
   S708_LM_DC_2ND_CLAMP3.Visu_Ret_Arr[1] := FALSE;
   S708_LM_DC_2ND_CLAMP3.Visu_Ret_Arr[2] := FALSE;
   S708_LM_DC_2ND_CLAMP3.Visu_Ret_Arr[3] := FALSE;
   S708_LM_DC_2ND_CLAMP3.Visu_Ret_Arr[4] := FALSE;
   S708_LM_DC_2ND_CLAMP3.Visu_Ret_Arr[5] := FALSE;
   S708_LM_DC_2ND_CLAMP3.Visu_Ret_Arr[6] := FALSE;
   S708_LM_DC_2ND_CLAMP3.Visu_Ret_Arr[7] := FALSE;
   S708_LM_DC_2ND_CLAMP3.Visu_Ret_Arr[8] := FALSE;
   S708_LM_DC_2ND_CLAMP3.Visu_Ret_Arr[9] := FALSE;
   S708_LM_DC_2ND_CLAMP3.Visu_Ret_Arr[10] := FALSE;
   S708_LM_DC_2ND_CLAMP3.Visu_Ret_Arr[11] := FALSE;
   S708_LM_DC_2ND_CLAMP3.Visu_Ret_Arr[12] := FALSE;
   S708_LM_DC_2ND_CLAMP3.Visu_Ret_Arr[13] := FALSE;
   S708_LM_DC_2ND_CLAMP3.Visu_Ret_Arr[14] := FALSE;
   S708_LM_DC_2ND_CLAMP3.Visu_Ret_Arr[15] := FALSE;
   S708_LM_DC_2ND_CLAMP3.BLK_Move_Ret := 0;
   S708_LM_DC_2ND_CLAMP3.Enable := FALSE;
   S708_LM_DC_2ND_CLAMP3.Adv_End := FALSE;
   S708_LM_DC_2ND_CLAMP3.Ret_End := FALSE;
   S708_LM_DC_2ND_CLAMP4.Enable_Aux := FALSE;
   S708_LM_DC_2ND_CLAMP4.Adv_Amount := 1;
   S708_LM_DC_2ND_CLAMP4.Ret_Amount := 1;
   S708_LM_DC_2ND_CLAMP4.LS_Adv1 := FALSE;
   S708_LM_DC_2ND_CLAMP4.LS_Ret1 := FALSE;
   S708_LM_DC_2ND_CLAMP4.LS_Adv2 := FALSE;
   S708_LM_DC_2ND_CLAMP4.LS_Ret2 := FALSE;
   S708_LM_DC_2ND_CLAMP4.LS_Adv3 := FALSE;
   S708_LM_DC_2ND_CLAMP4.LS_Ret3 := FALSE;
   S708_LM_DC_2ND_CLAMP4.LS_Adv4 := FALSE;
   S708_LM_DC_2ND_CLAMP4.LS_Ret4 := FALSE;
   S708_LM_DC_2ND_CLAMP4.SOL_Adv := FALSE;
   S708_LM_DC_2ND_CLAMP4.SOL_Ret := FALSE;
   S708_LM_DC_2ND_CLAMP4.M_Ready := TRUE;
   S708_LM_DC_2ND_CLAMP4.T_CHK1 := T#4S;
   S708_LM_DC_2ND_CLAMP4.T_CHK2 := T#4S;
   S708_LM_DC_2ND_CLAMP4.PB_Lamp_CHK := FALSE;
   S708_LM_DC_2ND_CLAMP4.PB_Error_Rst := FALSE;
   S708_LM_DC_2ND_CLAMP4.M_FLICK := TRUE;
   S708_LM_DC_2ND_CLAMP4.M_Adv_Err := FALSE;
   S708_LM_DC_2ND_CLAMP4.M_Ret_Err := FALSE;
   S708_LM_DC_2ND_CLAMP4.LP_Adv := FALSE;
   S708_LM_DC_2ND_CLAMP4.LP_Ret := FALSE;
   S708_LM_DC_2ND_CLAMP4.Visu_Adv := W#16#0;
   S708_LM_DC_2ND_CLAMP4.Visu_Ret := W#16#0;
   S708_LM_DC_2ND_CLAMP4.Error_T1.IN := FALSE;
   S708_LM_DC_2ND_CLAMP4.Error_T1.PT := T#4S;
   S708_LM_DC_2ND_CLAMP4.Error_T1.Q := FALSE;
   S708_LM_DC_2ND_CLAMP4.Error_T1.ET := T#0MS;
   S708_LM_DC_2ND_CLAMP4.Error_T1.STATE := B#16#0;
   S708_LM_DC_2ND_CLAMP4.Error_T1.STIME := T#0MS;
   S708_LM_DC_2ND_CLAMP4.Error_T1.ATIME := T#0MS;
   S708_LM_DC_2ND_CLAMP4.Error_T2.IN := FALSE;
   S708_LM_DC_2ND_CLAMP4.Error_T2.PT := T#4S;
   S708_LM_DC_2ND_CLAMP4.Error_T2.Q := FALSE;
   S708_LM_DC_2ND_CLAMP4.Error_T2.ET := T#0MS;
   S708_LM_DC_2ND_CLAMP4.Error_T2.STATE := B#16#0;
   S708_LM_DC_2ND_CLAMP4.Error_T2.STIME := T#0MS;
   S708_LM_DC_2ND_CLAMP4.Error_T2.ATIME := T#0MS;
   S708_LM_DC_2ND_CLAMP4.CHK_Aux1 := FALSE;
   S708_LM_DC_2ND_CLAMP4.CHK_Aux2 := FALSE;
   S708_LM_DC_2ND_CLAMP4.Error_T1_DN := FALSE;
   S708_LM_DC_2ND_CLAMP4.Error_T2_DN := FALSE;
   S708_LM_DC_2ND_CLAMP4.Adv_Memo := FALSE;
   S708_LM_DC_2ND_CLAMP4.Visu_Adv_Arr[0] := FALSE;
   S708_LM_DC_2ND_CLAMP4.Visu_Adv_Arr[1] := FALSE;
   S708_LM_DC_2ND_CLAMP4.Visu_Adv_Arr[2] := FALSE;
   S708_LM_DC_2ND_CLAMP4.Visu_Adv_Arr[3] := FALSE;
   S708_LM_DC_2ND_CLAMP4.Visu_Adv_Arr[4] := FALSE;
   S708_LM_DC_2ND_CLAMP4.Visu_Adv_Arr[5] := FALSE;
   S708_LM_DC_2ND_CLAMP4.Visu_Adv_Arr[6] := FALSE;
   S708_LM_DC_2ND_CLAMP4.Visu_Adv_Arr[7] := FALSE;
   S708_LM_DC_2ND_CLAMP4.Visu_Adv_Arr[8] := FALSE;
   S708_LM_DC_2ND_CLAMP4.Visu_Adv_Arr[9] := FALSE;
   S708_LM_DC_2ND_CLAMP4.Visu_Adv_Arr[10] := FALSE;
   S708_LM_DC_2ND_CLAMP4.Visu_Adv_Arr[11] := FALSE;
   S708_LM_DC_2ND_CLAMP4.Visu_Adv_Arr[12] := FALSE;
   S708_LM_DC_2ND_CLAMP4.Visu_Adv_Arr[13] := FALSE;
   S708_LM_DC_2ND_CLAMP4.Visu_Adv_Arr[14] := FALSE;
   S708_LM_DC_2ND_CLAMP4.Visu_Adv_Arr[15] := FALSE;
   S708_LM_DC_2ND_CLAMP4.Visu_Ret_Arr[0] := FALSE;
   S708_LM_DC_2ND_CLAMP4.Visu_Ret_Arr[1] := FALSE;
   S708_LM_DC_2ND_CLAMP4.Visu_Ret_Arr[2] := FALSE;
   S708_LM_DC_2ND_CLAMP4.Visu_Ret_Arr[3] := FALSE;
   S708_LM_DC_2ND_CLAMP4.Visu_Ret_Arr[4] := FALSE;
   S708_LM_DC_2ND_CLAMP4.Visu_Ret_Arr[5] := FALSE;
   S708_LM_DC_2ND_CLAMP4.Visu_Ret_Arr[6] := FALSE;
   S708_LM_DC_2ND_CLAMP4.Visu_Ret_Arr[7] := FALSE;
   S708_LM_DC_2ND_CLAMP4.Visu_Ret_Arr[8] := FALSE;
   S708_LM_DC_2ND_CLAMP4.Visu_Ret_Arr[9] := FALSE;
   S708_LM_DC_2ND_CLAMP4.Visu_Ret_Arr[10] := FALSE;
   S708_LM_DC_2ND_CLAMP4.Visu_Ret_Arr[11] := FALSE;
   S708_LM_DC_2ND_CLAMP4.Visu_Ret_Arr[12] := FALSE;
   S708_LM_DC_2ND_CLAMP4.Visu_Ret_Arr[13] := FALSE;
   S708_LM_DC_2ND_CLAMP4.Visu_Ret_Arr[14] := FALSE;
   S708_LM_DC_2ND_CLAMP4.Visu_Ret_Arr[15] := FALSE;
   S708_LM_DC_2ND_CLAMP4.BLK_Move_Ret := 0;
   S708_LM_DC_2ND_CLAMP4.Enable := FALSE;
   S708_LM_DC_2ND_CLAMP4.Adv_End := FALSE;
   S708_LM_DC_2ND_CLAMP4.Ret_End := FALSE;
   S708_LM_DC_2ND_CLAMP5.Enable_Aux := FALSE;
   S708_LM_DC_2ND_CLAMP5.Adv_Amount := 1;
   S708_LM_DC_2ND_CLAMP5.Ret_Amount := 1;
   S708_LM_DC_2ND_CLAMP5.LS_Adv1 := FALSE;
   S708_LM_DC_2ND_CLAMP5.LS_Ret1 := FALSE;
   S708_LM_DC_2ND_CLAMP5.LS_Adv2 := FALSE;
   S708_LM_DC_2ND_CLAMP5.LS_Ret2 := FALSE;
   S708_LM_DC_2ND_CLAMP5.LS_Adv3 := FALSE;
   S708_LM_DC_2ND_CLAMP5.LS_Ret3 := FALSE;
   S708_LM_DC_2ND_CLAMP5.LS_Adv4 := FALSE;
   S708_LM_DC_2ND_CLAMP5.LS_Ret4 := FALSE;
   S708_LM_DC_2ND_CLAMP5.SOL_Adv := FALSE;
   S708_LM_DC_2ND_CLAMP5.SOL_Ret := FALSE;
   S708_LM_DC_2ND_CLAMP5.M_Ready := TRUE;
   S708_LM_DC_2ND_CLAMP5.T_CHK1 := T#4S;
   S708_LM_DC_2ND_CLAMP5.T_CHK2 := T#4S;
   S708_LM_DC_2ND_CLAMP5.PB_Lamp_CHK := FALSE;
   S708_LM_DC_2ND_CLAMP5.PB_Error_Rst := FALSE;
   S708_LM_DC_2ND_CLAMP5.M_FLICK := TRUE;
   S708_LM_DC_2ND_CLAMP5.M_Adv_Err := FALSE;
   S708_LM_DC_2ND_CLAMP5.M_Ret_Err := FALSE;
   S708_LM_DC_2ND_CLAMP5.LP_Adv := FALSE;
   S708_LM_DC_2ND_CLAMP5.LP_Ret := FALSE;
   S708_LM_DC_2ND_CLAMP5.Visu_Adv := W#16#0;
   S708_LM_DC_2ND_CLAMP5.Visu_Ret := W#16#0;
   S708_LM_DC_2ND_CLAMP5.Error_T1.IN := FALSE;
   S708_LM_DC_2ND_CLAMP5.Error_T1.PT := T#4S;
   S708_LM_DC_2ND_CLAMP5.Error_T1.Q := FALSE;
   S708_LM_DC_2ND_CLAMP5.Error_T1.ET := T#0MS;
   S708_LM_DC_2ND_CLAMP5.Error_T1.STATE := B#16#0;
   S708_LM_DC_2ND_CLAMP5.Error_T1.STIME := T#0MS;
   S708_LM_DC_2ND_CLAMP5.Error_T1.ATIME := T#0MS;
   S708_LM_DC_2ND_CLAMP5.Error_T2.IN := FALSE;
   S708_LM_DC_2ND_CLAMP5.Error_T2.PT := T#4S;
   S708_LM_DC_2ND_CLAMP5.Error_T2.Q := FALSE;
   S708_LM_DC_2ND_CLAMP5.Error_T2.ET := T#0MS;
   S708_LM_DC_2ND_CLAMP5.Error_T2.STATE := B#16#0;
   S708_LM_DC_2ND_CLAMP5.Error_T2.STIME := T#0MS;
   S708_LM_DC_2ND_CLAMP5.Error_T2.ATIME := T#0MS;
   S708_LM_DC_2ND_CLAMP5.CHK_Aux1 := FALSE;
   S708_LM_DC_2ND_CLAMP5.CHK_Aux2 := FALSE;
   S708_LM_DC_2ND_CLAMP5.Error_T1_DN := FALSE;
   S708_LM_DC_2ND_CLAMP5.Error_T2_DN := FALSE;
   S708_LM_DC_2ND_CLAMP5.Adv_Memo := FALSE;
   S708_LM_DC_2ND_CLAMP5.Visu_Adv_Arr[0] := FALSE;
   S708_LM_DC_2ND_CLAMP5.Visu_Adv_Arr[1] := FALSE;
   S708_LM_DC_2ND_CLAMP5.Visu_Adv_Arr[2] := FALSE;
   S708_LM_DC_2ND_CLAMP5.Visu_Adv_Arr[3] := FALSE;
   S708_LM_DC_2ND_CLAMP5.Visu_Adv_Arr[4] := FALSE;
   S708_LM_DC_2ND_CLAMP5.Visu_Adv_Arr[5] := FALSE;
   S708_LM_DC_2ND_CLAMP5.Visu_Adv_Arr[6] := FALSE;
   S708_LM_DC_2ND_CLAMP5.Visu_Adv_Arr[7] := FALSE;
   S708_LM_DC_2ND_CLAMP5.Visu_Adv_Arr[8] := FALSE;
   S708_LM_DC_2ND_CLAMP5.Visu_Adv_Arr[9] := FALSE;
   S708_LM_DC_2ND_CLAMP5.Visu_Adv_Arr[10] := FALSE;
   S708_LM_DC_2ND_CLAMP5.Visu_Adv_Arr[11] := FALSE;
   S708_LM_DC_2ND_CLAMP5.Visu_Adv_Arr[12] := FALSE;
   S708_LM_DC_2ND_CLAMP5.Visu_Adv_Arr[13] := FALSE;
   S708_LM_DC_2ND_CLAMP5.Visu_Adv_Arr[14] := FALSE;
   S708_LM_DC_2ND_CLAMP5.Visu_Adv_Arr[15] := FALSE;
   S708_LM_DC_2ND_CLAMP5.Visu_Ret_Arr[0] := FALSE;
   S708_LM_DC_2ND_CLAMP5.Visu_Ret_Arr[1] := FALSE;
   S708_LM_DC_2ND_CLAMP5.Visu_Ret_Arr[2] := FALSE;
   S708_LM_DC_2ND_CLAMP5.Visu_Ret_Arr[3] := FALSE;
   S708_LM_DC_2ND_CLAMP5.Visu_Ret_Arr[4] := FALSE;
   S708_LM_DC_2ND_CLAMP5.Visu_Ret_Arr[5] := FALSE;
   S708_LM_DC_2ND_CLAMP5.Visu_Ret_Arr[6] := FALSE;
   S708_LM_DC_2ND_CLAMP5.Visu_Ret_Arr[7] := FALSE;
   S708_LM_DC_2ND_CLAMP5.Visu_Ret_Arr[8] := FALSE;
   S708_LM_DC_2ND_CLAMP5.Visu_Ret_Arr[9] := FALSE;
   S708_LM_DC_2ND_CLAMP5.Visu_Ret_Arr[10] := FALSE;
   S708_LM_DC_2ND_CLAMP5.Visu_Ret_Arr[11] := FALSE;
   S708_LM_DC_2ND_CLAMP5.Visu_Ret_Arr[12] := FALSE;
   S708_LM_DC_2ND_CLAMP5.Visu_Ret_Arr[13] := FALSE;
   S708_LM_DC_2ND_CLAMP5.Visu_Ret_Arr[14] := FALSE;
   S708_LM_DC_2ND_CLAMP5.Visu_Ret_Arr[15] := FALSE;
   S708_LM_DC_2ND_CLAMP5.BLK_Move_Ret := 0;
   S708_LM_DC_2ND_CLAMP5.Enable := FALSE;
   S708_LM_DC_2ND_CLAMP5.Adv_End := FALSE;
   S708_LM_DC_2ND_CLAMP5.Ret_End := FALSE;
   S708_LM_DC_STK_PIN.Enable_Aux := FALSE;
   S708_LM_DC_STK_PIN.Adv_Amount := 1;
   S708_LM_DC_STK_PIN.Ret_Amount := 1;
   S708_LM_DC_STK_PIN.LS_Adv1 := FALSE;
   S708_LM_DC_STK_PIN.LS_Ret1 := FALSE;
   S708_LM_DC_STK_PIN.LS_Adv2 := FALSE;
   S708_LM_DC_STK_PIN.LS_Ret2 := FALSE;
   S708_LM_DC_STK_PIN.LS_Adv3 := FALSE;
   S708_LM_DC_STK_PIN.LS_Ret3 := FALSE;
   S708_LM_DC_STK_PIN.LS_Adv4 := FALSE;
   S708_LM_DC_STK_PIN.LS_Ret4 := FALSE;
   S708_LM_DC_STK_PIN.SOL_Adv := FALSE;
   S708_LM_DC_STK_PIN.SOL_Ret := FALSE;
   S708_LM_DC_STK_PIN.M_Ready := TRUE;
   S708_LM_DC_STK_PIN.T_CHK1 := T#4S;
   S708_LM_DC_STK_PIN.T_CHK2 := T#4S;
   S708_LM_DC_STK_PIN.PB_Lamp_CHK := FALSE;
   S708_LM_DC_STK_PIN.PB_Error_Rst := FALSE;
   S708_LM_DC_STK_PIN.M_FLICK := TRUE;
   S708_LM_DC_STK_PIN.M_Adv_Err := FALSE;
   S708_LM_DC_STK_PIN.M_Ret_Err := FALSE;
   S708_LM_DC_STK_PIN.LP_Adv := FALSE;
   S708_LM_DC_STK_PIN.LP_Ret := FALSE;
   S708_LM_DC_STK_PIN.Visu_Adv := W#16#0;
   S708_LM_DC_STK_PIN.Visu_Ret := W#16#0;
   S708_LM_DC_STK_PIN.Error_T1.IN := FALSE;
   S708_LM_DC_STK_PIN.Error_T1.PT := T#4S;
   S708_LM_DC_STK_PIN.Error_T1.Q := FALSE;
   S708_LM_DC_STK_PIN.Error_T1.ET := T#0MS;
   S708_LM_DC_STK_PIN.Error_T1.STATE := B#16#0;
   S708_LM_DC_STK_PIN.Error_T1.STIME := T#0MS;
   S708_LM_DC_STK_PIN.Error_T1.ATIME := T#0MS;
   S708_LM_DC_STK_PIN.Error_T2.IN := FALSE;
   S708_LM_DC_STK_PIN.Error_T2.PT := T#4S;
   S708_LM_DC_STK_PIN.Error_T2.Q := FALSE;
   S708_LM_DC_STK_PIN.Error_T2.ET := T#0MS;
   S708_LM_DC_STK_PIN.Error_T2.STATE := B#16#0;
   S708_LM_DC_STK_PIN.Error_T2.STIME := T#0MS;
   S708_LM_DC_STK_PIN.Error_T2.ATIME := T#0MS;
   S708_LM_DC_STK_PIN.CHK_Aux1 := FALSE;
   S708_LM_DC_STK_PIN.CHK_Aux2 := FALSE;
   S708_LM_DC_STK_PIN.Error_T1_DN := FALSE;
   S708_LM_DC_STK_PIN.Error_T2_DN := FALSE;
   S708_LM_DC_STK_PIN.Adv_Memo := FALSE;
   S708_LM_DC_STK_PIN.Visu_Adv_Arr[0] := FALSE;
   S708_LM_DC_STK_PIN.Visu_Adv_Arr[1] := FALSE;
   S708_LM_DC_STK_PIN.Visu_Adv_Arr[2] := FALSE;
   S708_LM_DC_STK_PIN.Visu_Adv_Arr[3] := FALSE;
   S708_LM_DC_STK_PIN.Visu_Adv_Arr[4] := FALSE;
   S708_LM_DC_STK_PIN.Visu_Adv_Arr[5] := FALSE;
   S708_LM_DC_STK_PIN.Visu_Adv_Arr[6] := FALSE;
   S708_LM_DC_STK_PIN.Visu_Adv_Arr[7] := FALSE;
   S708_LM_DC_STK_PIN.Visu_Adv_Arr[8] := FALSE;
   S708_LM_DC_STK_PIN.Visu_Adv_Arr[9] := FALSE;
   S708_LM_DC_STK_PIN.Visu_Adv_Arr[10] := FALSE;
   S708_LM_DC_STK_PIN.Visu_Adv_Arr[11] := FALSE;
   S708_LM_DC_STK_PIN.Visu_Adv_Arr[12] := FALSE;
   S708_LM_DC_STK_PIN.Visu_Adv_Arr[13] := FALSE;
   S708_LM_DC_STK_PIN.Visu_Adv_Arr[14] := FALSE;
   S708_LM_DC_STK_PIN.Visu_Adv_Arr[15] := FALSE;
   S708_LM_DC_STK_PIN.Visu_Ret_Arr[0] := FALSE;
   S708_LM_DC_STK_PIN.Visu_Ret_Arr[1] := FALSE;
   S708_LM_DC_STK_PIN.Visu_Ret_Arr[2] := FALSE;
   S708_LM_DC_STK_PIN.Visu_Ret_Arr[3] := FALSE;
   S708_LM_DC_STK_PIN.Visu_Ret_Arr[4] := FALSE;
   S708_LM_DC_STK_PIN.Visu_Ret_Arr[5] := FALSE;
   S708_LM_DC_STK_PIN.Visu_Ret_Arr[6] := FALSE;
   S708_LM_DC_STK_PIN.Visu_Ret_Arr[7] := FALSE;
   S708_LM_DC_STK_PIN.Visu_Ret_Arr[8] := FALSE;
   S708_LM_DC_STK_PIN.Visu_Ret_Arr[9] := FALSE;
   S708_LM_DC_STK_PIN.Visu_Ret_Arr[10] := FALSE;
   S708_LM_DC_STK_PIN.Visu_Ret_Arr[11] := FALSE;
   S708_LM_DC_STK_PIN.Visu_Ret_Arr[12] := FALSE;
   S708_LM_DC_STK_PIN.Visu_Ret_Arr[13] := FALSE;
   S708_LM_DC_STK_PIN.Visu_Ret_Arr[14] := FALSE;
   S708_LM_DC_STK_PIN.Visu_Ret_Arr[15] := FALSE;
   S708_LM_DC_STK_PIN.BLK_Move_Ret := 0;
   S708_LM_DC_STK_PIN.Enable := FALSE;
   S708_LM_DC_STK_PIN.Adv_End := FALSE;
   S708_LM_DC_STK_PIN.Ret_End := FALSE;
   S708_LM_DC_OTR_CLAMP.Enable_Aux := FALSE;
   S708_LM_DC_OTR_CLAMP.Adv_Amount := 1;
   S708_LM_DC_OTR_CLAMP.Ret_Amount := 1;
   S708_LM_DC_OTR_CLAMP.LS_Adv1 := FALSE;
   S708_LM_DC_OTR_CLAMP.LS_Ret1 := FALSE;
   S708_LM_DC_OTR_CLAMP.LS_Adv2 := FALSE;
   S708_LM_DC_OTR_CLAMP.LS_Ret2 := FALSE;
   S708_LM_DC_OTR_CLAMP.LS_Adv3 := FALSE;
   S708_LM_DC_OTR_CLAMP.LS_Ret3 := FALSE;
   S708_LM_DC_OTR_CLAMP.LS_Adv4 := FALSE;
   S708_LM_DC_OTR_CLAMP.LS_Ret4 := FALSE;
   S708_LM_DC_OTR_CLAMP.SOL_Adv := FALSE;
   S708_LM_DC_OTR_CLAMP.SOL_Ret := FALSE;
   S708_LM_DC_OTR_CLAMP.M_Ready := TRUE;
   S708_LM_DC_OTR_CLAMP.T_CHK1 := T#4S;
   S708_LM_DC_OTR_CLAMP.T_CHK2 := T#4S;
   S708_LM_DC_OTR_CLAMP.PB_Lamp_CHK := FALSE;
   S708_LM_DC_OTR_CLAMP.PB_Error_Rst := FALSE;
   S708_LM_DC_OTR_CLAMP.M_FLICK := TRUE;
   S708_LM_DC_OTR_CLAMP.M_Adv_Err := FALSE;
   S708_LM_DC_OTR_CLAMP.M_Ret_Err := FALSE;
   S708_LM_DC_OTR_CLAMP.LP_Adv := FALSE;
   S708_LM_DC_OTR_CLAMP.LP_Ret := FALSE;
   S708_LM_DC_OTR_CLAMP.Visu_Adv := W#16#0;
   S708_LM_DC_OTR_CLAMP.Visu_Ret := W#16#0;
   S708_LM_DC_OTR_CLAMP.Error_T1.IN := FALSE;
   S708_LM_DC_OTR_CLAMP.Error_T1.PT := T#4S;
   S708_LM_DC_OTR_CLAMP.Error_T1.Q := FALSE;
   S708_LM_DC_OTR_CLAMP.Error_T1.ET := T#0MS;
   S708_LM_DC_OTR_CLAMP.Error_T1.STATE := B#16#0;
   S708_LM_DC_OTR_CLAMP.Error_T1.STIME := T#0MS;
   S708_LM_DC_OTR_CLAMP.Error_T1.ATIME := T#0MS;
   S708_LM_DC_OTR_CLAMP.Error_T2.IN := FALSE;
   S708_LM_DC_OTR_CLAMP.Error_T2.PT := T#4S;
   S708_LM_DC_OTR_CLAMP.Error_T2.Q := FALSE;
   S708_LM_DC_OTR_CLAMP.Error_T2.ET := T#0MS;
   S708_LM_DC_OTR_CLAMP.Error_T2.STATE := B#16#0;
   S708_LM_DC_OTR_CLAMP.Error_T2.STIME := T#0MS;
   S708_LM_DC_OTR_CLAMP.Error_T2.ATIME := T#0MS;
   S708_LM_DC_OTR_CLAMP.CHK_Aux1 := FALSE;
   S708_LM_DC_OTR_CLAMP.CHK_Aux2 := FALSE;
   S708_LM_DC_OTR_CLAMP.Error_T1_DN := FALSE;
   S708_LM_DC_OTR_CLAMP.Error_T2_DN := FALSE;
   S708_LM_DC_OTR_CLAMP.Adv_Memo := FALSE;
   S708_LM_DC_OTR_CLAMP.Visu_Adv_Arr[0] := FALSE;
   S708_LM_DC_OTR_CLAMP.Visu_Adv_Arr[1] := FALSE;
   S708_LM_DC_OTR_CLAMP.Visu_Adv_Arr[2] := FALSE;
   S708_LM_DC_OTR_CLAMP.Visu_Adv_Arr[3] := FALSE;
   S708_LM_DC_OTR_CLAMP.Visu_Adv_Arr[4] := FALSE;
   S708_LM_DC_OTR_CLAMP.Visu_Adv_Arr[5] := FALSE;
   S708_LM_DC_OTR_CLAMP.Visu_Adv_Arr[6] := FALSE;
   S708_LM_DC_OTR_CLAMP.Visu_Adv_Arr[7] := FALSE;
   S708_LM_DC_OTR_CLAMP.Visu_Adv_Arr[8] := FALSE;
   S708_LM_DC_OTR_CLAMP.Visu_Adv_Arr[9] := FALSE;
   S708_LM_DC_OTR_CLAMP.Visu_Adv_Arr[10] := FALSE;
   S708_LM_DC_OTR_CLAMP.Visu_Adv_Arr[11] := FALSE;
   S708_LM_DC_OTR_CLAMP.Visu_Adv_Arr[12] := FALSE;
   S708_LM_DC_OTR_CLAMP.Visu_Adv_Arr[13] := FALSE;
   S708_LM_DC_OTR_CLAMP.Visu_Adv_Arr[14] := FALSE;
   S708_LM_DC_OTR_CLAMP.Visu_Adv_Arr[15] := FALSE;
   S708_LM_DC_OTR_CLAMP.Visu_Ret_Arr[0] := FALSE;
   S708_LM_DC_OTR_CLAMP.Visu_Ret_Arr[1] := FALSE;
   S708_LM_DC_OTR_CLAMP.Visu_Ret_Arr[2] := FALSE;
   S708_LM_DC_OTR_CLAMP.Visu_Ret_Arr[3] := FALSE;
   S708_LM_DC_OTR_CLAMP.Visu_Ret_Arr[4] := FALSE;
   S708_LM_DC_OTR_CLAMP.Visu_Ret_Arr[5] := FALSE;
   S708_LM_DC_OTR_CLAMP.Visu_Ret_Arr[6] := FALSE;
   S708_LM_DC_OTR_CLAMP.Visu_Ret_Arr[7] := FALSE;
   S708_LM_DC_OTR_CLAMP.Visu_Ret_Arr[8] := FALSE;
   S708_LM_DC_OTR_CLAMP.Visu_Ret_Arr[9] := FALSE;
   S708_LM_DC_OTR_CLAMP.Visu_Ret_Arr[10] := FALSE;
   S708_LM_DC_OTR_CLAMP.Visu_Ret_Arr[11] := FALSE;
   S708_LM_DC_OTR_CLAMP.Visu_Ret_Arr[12] := FALSE;
   S708_LM_DC_OTR_CLAMP.Visu_Ret_Arr[13] := FALSE;
   S708_LM_DC_OTR_CLAMP.Visu_Ret_Arr[14] := FALSE;
   S708_LM_DC_OTR_CLAMP.Visu_Ret_Arr[15] := FALSE;
   S708_LM_DC_OTR_CLAMP.BLK_Move_Ret := 0;
   S708_LM_DC_OTR_CLAMP.Enable := FALSE;
   S708_LM_DC_OTR_CLAMP.Adv_End := FALSE;
   S708_LM_DC_OTR_CLAMP.Ret_End := FALSE;
   S708_LM_DC_ASSY_CLAMP.Enable_Aux := FALSE;
   S708_LM_DC_ASSY_CLAMP.Adv_Amount := 1;
   S708_LM_DC_ASSY_CLAMP.Ret_Amount := 1;
   S708_LM_DC_ASSY_CLAMP.LS_Adv1 := FALSE;
   S708_LM_DC_ASSY_CLAMP.LS_Ret1 := FALSE;
   S708_LM_DC_ASSY_CLAMP.LS_Adv2 := FALSE;
   S708_LM_DC_ASSY_CLAMP.LS_Ret2 := FALSE;
   S708_LM_DC_ASSY_CLAMP.LS_Adv3 := FALSE;
   S708_LM_DC_ASSY_CLAMP.LS_Ret3 := FALSE;
   S708_LM_DC_ASSY_CLAMP.LS_Adv4 := FALSE;
   S708_LM_DC_ASSY_CLAMP.LS_Ret4 := FALSE;
   S708_LM_DC_ASSY_CLAMP.SOL_Adv := FALSE;
   S708_LM_DC_ASSY_CLAMP.SOL_Ret := FALSE;
   S708_LM_DC_ASSY_CLAMP.M_Ready := TRUE;
   S708_LM_DC_ASSY_CLAMP.T_CHK1 := T#4S;
   S708_LM_DC_ASSY_CLAMP.T_CHK2 := T#4S;
   S708_LM_DC_ASSY_CLAMP.PB_Lamp_CHK := FALSE;
   S708_LM_DC_ASSY_CLAMP.PB_Error_Rst := FALSE;
   S708_LM_DC_ASSY_CLAMP.M_FLICK := TRUE;
   S708_LM_DC_ASSY_CLAMP.M_Adv_Err := FALSE;
   S708_LM_DC_ASSY_CLAMP.M_Ret_Err := FALSE;
   S708_LM_DC_ASSY_CLAMP.LP_Adv := FALSE;
   S708_LM_DC_ASSY_CLAMP.LP_Ret := FALSE;
   S708_LM_DC_ASSY_CLAMP.Visu_Adv := W#16#0;
   S708_LM_DC_ASSY_CLAMP.Visu_Ret := W#16#0;
   S708_LM_DC_ASSY_CLAMP.Error_T1.IN := FALSE;
   S708_LM_DC_ASSY_CLAMP.Error_T1.PT := T#4S;
   S708_LM_DC_ASSY_CLAMP.Error_T1.Q := FALSE;
   S708_LM_DC_ASSY_CLAMP.Error_T1.ET := T#0MS;
   S708_LM_DC_ASSY_CLAMP.Error_T1.STATE := B#16#0;
   S708_LM_DC_ASSY_CLAMP.Error_T1.STIME := T#22D23H1M2S541MS;
   S708_LM_DC_ASSY_CLAMP.Error_T1.ATIME := T#22D23H1M3S288MS;
   S708_LM_DC_ASSY_CLAMP.Error_T2.IN := FALSE;
   S708_LM_DC_ASSY_CLAMP.Error_T2.PT := T#4S;
   S708_LM_DC_ASSY_CLAMP.Error_T2.Q := FALSE;
   S708_LM_DC_ASSY_CLAMP.Error_T2.ET := T#0MS;
   S708_LM_DC_ASSY_CLAMP.Error_T2.STATE := B#16#0;
   S708_LM_DC_ASSY_CLAMP.Error_T2.STIME := T#0MS;
   S708_LM_DC_ASSY_CLAMP.Error_T2.ATIME := T#0MS;
   S708_LM_DC_ASSY_CLAMP.CHK_Aux1 := FALSE;
   S708_LM_DC_ASSY_CLAMP.CHK_Aux2 := FALSE;
   S708_LM_DC_ASSY_CLAMP.Error_T1_DN := FALSE;
   S708_LM_DC_ASSY_CLAMP.Error_T2_DN := FALSE;
   S708_LM_DC_ASSY_CLAMP.Adv_Memo := FALSE;
   S708_LM_DC_ASSY_CLAMP.Visu_Adv_Arr[0] := FALSE;
   S708_LM_DC_ASSY_CLAMP.Visu_Adv_Arr[1] := FALSE;
   S708_LM_DC_ASSY_CLAMP.Visu_Adv_Arr[2] := FALSE;
   S708_LM_DC_ASSY_CLAMP.Visu_Adv_Arr[3] := FALSE;
   S708_LM_DC_ASSY_CLAMP.Visu_Adv_Arr[4] := FALSE;
   S708_LM_DC_ASSY_CLAMP.Visu_Adv_Arr[5] := FALSE;
   S708_LM_DC_ASSY_CLAMP.Visu_Adv_Arr[6] := FALSE;
   S708_LM_DC_ASSY_CLAMP.Visu_Adv_Arr[7] := FALSE;
   S708_LM_DC_ASSY_CLAMP.Visu_Adv_Arr[8] := FALSE;
   S708_LM_DC_ASSY_CLAMP.Visu_Adv_Arr[9] := FALSE;
   S708_LM_DC_ASSY_CLAMP.Visu_Adv_Arr[10] := FALSE;
   S708_LM_DC_ASSY_CLAMP.Visu_Adv_Arr[11] := FALSE;
   S708_LM_DC_ASSY_CLAMP.Visu_Adv_Arr[12] := FALSE;
   S708_LM_DC_ASSY_CLAMP.Visu_Adv_Arr[13] := FALSE;
   S708_LM_DC_ASSY_CLAMP.Visu_Adv_Arr[14] := FALSE;
   S708_LM_DC_ASSY_CLAMP.Visu_Adv_Arr[15] := FALSE;
   S708_LM_DC_ASSY_CLAMP.Visu_Ret_Arr[0] := FALSE;
   S708_LM_DC_ASSY_CLAMP.Visu_Ret_Arr[1] := FALSE;
   S708_LM_DC_ASSY_CLAMP.Visu_Ret_Arr[2] := FALSE;
   S708_LM_DC_ASSY_CLAMP.Visu_Ret_Arr[3] := FALSE;
   S708_LM_DC_ASSY_CLAMP.Visu_Ret_Arr[4] := FALSE;
   S708_LM_DC_ASSY_CLAMP.Visu_Ret_Arr[5] := FALSE;
   S708_LM_DC_ASSY_CLAMP.Visu_Ret_Arr[6] := FALSE;
   S708_LM_DC_ASSY_CLAMP.Visu_Ret_Arr[7] := FALSE;
   S708_LM_DC_ASSY_CLAMP.Visu_Ret_Arr[8] := FALSE;
   S708_LM_DC_ASSY_CLAMP.Visu_Ret_Arr[9] := FALSE;
   S708_LM_DC_ASSY_CLAMP.Visu_Ret_Arr[10] := FALSE;
   S708_LM_DC_ASSY_CLAMP.Visu_Ret_Arr[11] := FALSE;
   S708_LM_DC_ASSY_CLAMP.Visu_Ret_Arr[12] := FALSE;
   S708_LM_DC_ASSY_CLAMP.Visu_Ret_Arr[13] := FALSE;
   S708_LM_DC_ASSY_CLAMP.Visu_Ret_Arr[14] := FALSE;
   S708_LM_DC_ASSY_CLAMP.Visu_Ret_Arr[15] := FALSE;
   S708_LM_DC_ASSY_CLAMP.BLK_Move_Ret := 0;
   S708_LM_DC_ASSY_CLAMP.Enable := FALSE;
   S708_LM_DC_ASSY_CLAMP.Adv_End := FALSE;
   S708_LM_DC_ASSY_CLAMP.Ret_End := FALSE;
   S708_LM_DC_FF_PIN.Enable_Aux := FALSE;
   S708_LM_DC_FF_PIN.Adv_Amount := 1;
   S708_LM_DC_FF_PIN.Ret_Amount := 1;
   S708_LM_DC_FF_PIN.LS_Adv1 := FALSE;
   S708_LM_DC_FF_PIN.LS_Ret1 := FALSE;
   S708_LM_DC_FF_PIN.LS_Adv2 := FALSE;
   S708_LM_DC_FF_PIN.LS_Ret2 := FALSE;
   S708_LM_DC_FF_PIN.LS_Adv3 := FALSE;
   S708_LM_DC_FF_PIN.LS_Ret3 := FALSE;
   S708_LM_DC_FF_PIN.LS_Adv4 := FALSE;
   S708_LM_DC_FF_PIN.LS_Ret4 := FALSE;
   S708_LM_DC_FF_PIN.SOL_Adv := FALSE;
   S708_LM_DC_FF_PIN.SOL_Ret := FALSE;
   S708_LM_DC_FF_PIN.M_Ready := TRUE;
   S708_LM_DC_FF_PIN.T_CHK1 := T#4S;
   S708_LM_DC_FF_PIN.T_CHK2 := T#4S;
   S708_LM_DC_FF_PIN.PB_Lamp_CHK := FALSE;
   S708_LM_DC_FF_PIN.PB_Error_Rst := FALSE;
   S708_LM_DC_FF_PIN.M_FLICK := TRUE;
   S708_LM_DC_FF_PIN.M_Adv_Err := FALSE;
   S708_LM_DC_FF_PIN.M_Ret_Err := FALSE;
   S708_LM_DC_FF_PIN.LP_Adv := FALSE;
   S708_LM_DC_FF_PIN.LP_Ret := FALSE;
   S708_LM_DC_FF_PIN.Visu_Adv := W#16#0;
   S708_LM_DC_FF_PIN.Visu_Ret := W#16#0;
   S708_LM_DC_FF_PIN.Error_T1.IN := FALSE;
   S708_LM_DC_FF_PIN.Error_T1.PT := T#4S;
   S708_LM_DC_FF_PIN.Error_T1.Q := FALSE;
   S708_LM_DC_FF_PIN.Error_T1.ET := T#0MS;
   S708_LM_DC_FF_PIN.Error_T1.STATE := B#16#0;
   S708_LM_DC_FF_PIN.Error_T1.STIME := T#4D10H46M40S935MS;
   S708_LM_DC_FF_PIN.Error_T1.ATIME := T#4D10H46M41S186MS;
   S708_LM_DC_FF_PIN.Error_T2.IN := FALSE;
   S708_LM_DC_FF_PIN.Error_T2.PT := T#4S;
   S708_LM_DC_FF_PIN.Error_T2.Q := FALSE;
   S708_LM_DC_FF_PIN.Error_T2.ET := T#0MS;
   S708_LM_DC_FF_PIN.Error_T2.STATE := B#16#0;
   S708_LM_DC_FF_PIN.Error_T2.STIME := T#0MS;
   S708_LM_DC_FF_PIN.Error_T2.ATIME := T#0MS;
   S708_LM_DC_FF_PIN.CHK_Aux1 := FALSE;
   S708_LM_DC_FF_PIN.CHK_Aux2 := FALSE;
   S708_LM_DC_FF_PIN.Error_T1_DN := FALSE;
   S708_LM_DC_FF_PIN.Error_T2_DN := FALSE;
   S708_LM_DC_FF_PIN.Adv_Memo := FALSE;
   S708_LM_DC_FF_PIN.Visu_Adv_Arr[0] := FALSE;
   S708_LM_DC_FF_PIN.Visu_Adv_Arr[1] := FALSE;
   S708_LM_DC_FF_PIN.Visu_Adv_Arr[2] := FALSE;
   S708_LM_DC_FF_PIN.Visu_Adv_Arr[3] := FALSE;
   S708_LM_DC_FF_PIN.Visu_Adv_Arr[4] := FALSE;
   S708_LM_DC_FF_PIN.Visu_Adv_Arr[5] := FALSE;
   S708_LM_DC_FF_PIN.Visu_Adv_Arr[6] := FALSE;
   S708_LM_DC_FF_PIN.Visu_Adv_Arr[7] := FALSE;
   S708_LM_DC_FF_PIN.Visu_Adv_Arr[8] := FALSE;
   S708_LM_DC_FF_PIN.Visu_Adv_Arr[9] := FALSE;
   S708_LM_DC_FF_PIN.Visu_Adv_Arr[10] := FALSE;
   S708_LM_DC_FF_PIN.Visu_Adv_Arr[11] := FALSE;
   S708_LM_DC_FF_PIN.Visu_Adv_Arr[12] := FALSE;
   S708_LM_DC_FF_PIN.Visu_Adv_Arr[13] := FALSE;
   S708_LM_DC_FF_PIN.Visu_Adv_Arr[14] := FALSE;
   S708_LM_DC_FF_PIN.Visu_Adv_Arr[15] := FALSE;
   S708_LM_DC_FF_PIN.Visu_Ret_Arr[0] := FALSE;
   S708_LM_DC_FF_PIN.Visu_Ret_Arr[1] := FALSE;
   S708_LM_DC_FF_PIN.Visu_Ret_Arr[2] := FALSE;
   S708_LM_DC_FF_PIN.Visu_Ret_Arr[3] := FALSE;
   S708_LM_DC_FF_PIN.Visu_Ret_Arr[4] := FALSE;
   S708_LM_DC_FF_PIN.Visu_Ret_Arr[5] := FALSE;
   S708_LM_DC_FF_PIN.Visu_Ret_Arr[6] := FALSE;
   S708_LM_DC_FF_PIN.Visu_Ret_Arr[7] := FALSE;
   S708_LM_DC_FF_PIN.Visu_Ret_Arr[8] := FALSE;
   S708_LM_DC_FF_PIN.Visu_Ret_Arr[9] := FALSE;
   S708_LM_DC_FF_PIN.Visu_Ret_Arr[10] := FALSE;
   S708_LM_DC_FF_PIN.Visu_Ret_Arr[11] := FALSE;
   S708_LM_DC_FF_PIN.Visu_Ret_Arr[12] := FALSE;
   S708_LM_DC_FF_PIN.Visu_Ret_Arr[13] := FALSE;
   S708_LM_DC_FF_PIN.Visu_Ret_Arr[14] := FALSE;
   S708_LM_DC_FF_PIN.Visu_Ret_Arr[15] := FALSE;
   S708_LM_DC_FF_PIN.BLK_Move_Ret := 0;
   S708_LM_DC_FF_PIN.Enable := FALSE;
   S708_LM_DC_FF_PIN.Adv_End := FALSE;
   S708_LM_DC_FF_PIN.Ret_End := FALSE;
   S708_LM_DC_FF_CLAMP.Enable_Aux := FALSE;
   S708_LM_DC_FF_CLAMP.Adv_Amount := 1;
   S708_LM_DC_FF_CLAMP.Ret_Amount := 1;
   S708_LM_DC_FF_CLAMP.LS_Adv1 := FALSE;
   S708_LM_DC_FF_CLAMP.LS_Ret1 := FALSE;
   S708_LM_DC_FF_CLAMP.LS_Adv2 := FALSE;
   S708_LM_DC_FF_CLAMP.LS_Ret2 := FALSE;
   S708_LM_DC_FF_CLAMP.LS_Adv3 := FALSE;
   S708_LM_DC_FF_CLAMP.LS_Ret3 := FALSE;
   S708_LM_DC_FF_CLAMP.LS_Adv4 := FALSE;
   S708_LM_DC_FF_CLAMP.LS_Ret4 := FALSE;
   S708_LM_DC_FF_CLAMP.SOL_Adv := FALSE;
   S708_LM_DC_FF_CLAMP.SOL_Ret := FALSE;
   S708_LM_DC_FF_CLAMP.M_Ready := TRUE;
   S708_LM_DC_FF_CLAMP.T_CHK1 := T#4S;
   S708_LM_DC_FF_CLAMP.T_CHK2 := T#4S;
   S708_LM_DC_FF_CLAMP.PB_Lamp_CHK := FALSE;
   S708_LM_DC_FF_CLAMP.PB_Error_Rst := FALSE;
   S708_LM_DC_FF_CLAMP.M_FLICK := TRUE;
   S708_LM_DC_FF_CLAMP.M_Adv_Err := FALSE;
   S708_LM_DC_FF_CLAMP.M_Ret_Err := FALSE;
   S708_LM_DC_FF_CLAMP.LP_Adv := FALSE;
   S708_LM_DC_FF_CLAMP.LP_Ret := FALSE;
   S708_LM_DC_FF_CLAMP.Visu_Adv := W#16#0;
   S708_LM_DC_FF_CLAMP.Visu_Ret := W#16#0;
   S708_LM_DC_FF_CLAMP.Error_T1.IN := FALSE;
   S708_LM_DC_FF_CLAMP.Error_T1.PT := T#4S;
   S708_LM_DC_FF_CLAMP.Error_T1.Q := FALSE;
   S708_LM_DC_FF_CLAMP.Error_T1.ET := T#0MS;
   S708_LM_DC_FF_CLAMP.Error_T1.STATE := B#16#0;
   S708_LM_DC_FF_CLAMP.Error_T1.STIME := T#4D10H46M40S935MS;
   S708_LM_DC_FF_CLAMP.Error_T1.ATIME := T#4D10H46M41S916MS;
   S708_LM_DC_FF_CLAMP.Error_T2.IN := FALSE;
   S708_LM_DC_FF_CLAMP.Error_T2.PT := T#4S;
   S708_LM_DC_FF_CLAMP.Error_T2.Q := FALSE;
   S708_LM_DC_FF_CLAMP.Error_T2.ET := T#0MS;
   S708_LM_DC_FF_CLAMP.Error_T2.STATE := B#16#0;
   S708_LM_DC_FF_CLAMP.Error_T2.STIME := T#0MS;
   S708_LM_DC_FF_CLAMP.Error_T2.ATIME := T#0MS;
   S708_LM_DC_FF_CLAMP.CHK_Aux1 := FALSE;
   S708_LM_DC_FF_CLAMP.CHK_Aux2 := FALSE;
   S708_LM_DC_FF_CLAMP.Error_T1_DN := FALSE;
   S708_LM_DC_FF_CLAMP.Error_T2_DN := FALSE;
   S708_LM_DC_FF_CLAMP.Adv_Memo := FALSE;
   S708_LM_DC_FF_CLAMP.Visu_Adv_Arr[0] := FALSE;
   S708_LM_DC_FF_CLAMP.Visu_Adv_Arr[1] := FALSE;
   S708_LM_DC_FF_CLAMP.Visu_Adv_Arr[2] := FALSE;
   S708_LM_DC_FF_CLAMP.Visu_Adv_Arr[3] := FALSE;
   S708_LM_DC_FF_CLAMP.Visu_Adv_Arr[4] := FALSE;
   S708_LM_DC_FF_CLAMP.Visu_Adv_Arr[5] := FALSE;
   S708_LM_DC_FF_CLAMP.Visu_Adv_Arr[6] := FALSE;
   S708_LM_DC_FF_CLAMP.Visu_Adv_Arr[7] := FALSE;
   S708_LM_DC_FF_CLAMP.Visu_Adv_Arr[8] := FALSE;
   S708_LM_DC_FF_CLAMP.Visu_Adv_Arr[9] := FALSE;
   S708_LM_DC_FF_CLAMP.Visu_Adv_Arr[10] := FALSE;
   S708_LM_DC_FF_CLAMP.Visu_Adv_Arr[11] := FALSE;
   S708_LM_DC_FF_CLAMP.Visu_Adv_Arr[12] := FALSE;
   S708_LM_DC_FF_CLAMP.Visu_Adv_Arr[13] := FALSE;
   S708_LM_DC_FF_CLAMP.Visu_Adv_Arr[14] := FALSE;
   S708_LM_DC_FF_CLAMP.Visu_Adv_Arr[15] := FALSE;
   S708_LM_DC_FF_CLAMP.Visu_Ret_Arr[0] := FALSE;
   S708_LM_DC_FF_CLAMP.Visu_Ret_Arr[1] := FALSE;
   S708_LM_DC_FF_CLAMP.Visu_Ret_Arr[2] := FALSE;
   S708_LM_DC_FF_CLAMP.Visu_Ret_Arr[3] := FALSE;
   S708_LM_DC_FF_CLAMP.Visu_Ret_Arr[4] := FALSE;
   S708_LM_DC_FF_CLAMP.Visu_Ret_Arr[5] := FALSE;
   S708_LM_DC_FF_CLAMP.Visu_Ret_Arr[6] := FALSE;
   S708_LM_DC_FF_CLAMP.Visu_Ret_Arr[7] := FALSE;
   S708_LM_DC_FF_CLAMP.Visu_Ret_Arr[8] := FALSE;
   S708_LM_DC_FF_CLAMP.Visu_Ret_Arr[9] := FALSE;
   S708_LM_DC_FF_CLAMP.Visu_Ret_Arr[10] := FALSE;
   S708_LM_DC_FF_CLAMP.Visu_Ret_Arr[11] := FALSE;
   S708_LM_DC_FF_CLAMP.Visu_Ret_Arr[12] := FALSE;
   S708_LM_DC_FF_CLAMP.Visu_Ret_Arr[13] := FALSE;
   S708_LM_DC_FF_CLAMP.Visu_Ret_Arr[14] := FALSE;
   S708_LM_DC_FF_CLAMP.Visu_Ret_Arr[15] := FALSE;
   S708_LM_DC_FF_CLAMP.BLK_Move_Ret := 0;
   S708_LM_DC_FF_CLAMP.Enable := FALSE;
   S708_LM_DC_FF_CLAMP.Adv_End := FALSE;
   S708_LM_DC_FF_CLAMP.Ret_End := FALSE;
   S708_LM_DC_2ND_CLAMP6.Enable_Aux := FALSE;
   S708_LM_DC_2ND_CLAMP6.Adv_Amount := 2;
   S708_LM_DC_2ND_CLAMP6.Ret_Amount := 2;
   S708_LM_DC_2ND_CLAMP6.LS_Adv1 := FALSE;
   S708_LM_DC_2ND_CLAMP6.LS_Ret1 := FALSE;
   S708_LM_DC_2ND_CLAMP6.LS_Adv2 := FALSE;
   S708_LM_DC_2ND_CLAMP6.LS_Ret2 := FALSE;
   S708_LM_DC_2ND_CLAMP6.LS_Adv3 := FALSE;
   S708_LM_DC_2ND_CLAMP6.LS_Ret3 := FALSE;
   S708_LM_DC_2ND_CLAMP6.LS_Adv4 := FALSE;
   S708_LM_DC_2ND_CLAMP6.LS_Ret4 := FALSE;
   S708_LM_DC_2ND_CLAMP6.SOL_Adv := FALSE;
   S708_LM_DC_2ND_CLAMP6.SOL_Ret := FALSE;
   S708_LM_DC_2ND_CLAMP6.M_Ready := TRUE;
   S708_LM_DC_2ND_CLAMP6.T_CHK1 := T#4S;
   S708_LM_DC_2ND_CLAMP6.T_CHK2 := T#4S;
   S708_LM_DC_2ND_CLAMP6.PB_Lamp_CHK := FALSE;
   S708_LM_DC_2ND_CLAMP6.PB_Error_Rst := FALSE;
   S708_LM_DC_2ND_CLAMP6.M_FLICK := TRUE;
   S708_LM_DC_2ND_CLAMP6.M_Adv_Err := FALSE;
   S708_LM_DC_2ND_CLAMP6.M_Ret_Err := FALSE;
   S708_LM_DC_2ND_CLAMP6.LP_Adv := FALSE;
   S708_LM_DC_2ND_CLAMP6.LP_Ret := FALSE;
   S708_LM_DC_2ND_CLAMP6.Visu_Adv := W#16#0;
   S708_LM_DC_2ND_CLAMP6.Visu_Ret := W#16#0;
   S708_LM_DC_2ND_CLAMP6.Error_T1.IN := FALSE;
   S708_LM_DC_2ND_CLAMP6.Error_T1.PT := T#4S;
   S708_LM_DC_2ND_CLAMP6.Error_T1.Q := FALSE;
   S708_LM_DC_2ND_CLAMP6.Error_T1.ET := T#0MS;
   S708_LM_DC_2ND_CLAMP6.Error_T1.STATE := B#16#0;
   S708_LM_DC_2ND_CLAMP6.Error_T1.STIME := T#22D23H1M2S541MS;
   S708_LM_DC_2ND_CLAMP6.Error_T1.ATIME := T#22D23H1M3S514MS;
   S708_LM_DC_2ND_CLAMP6.Error_T2.IN := FALSE;
   S708_LM_DC_2ND_CLAMP6.Error_T2.PT := T#4S;
   S708_LM_DC_2ND_CLAMP6.Error_T2.Q := FALSE;
   S708_LM_DC_2ND_CLAMP6.Error_T2.ET := T#0MS;
   S708_LM_DC_2ND_CLAMP6.Error_T2.STATE := B#16#0;
   S708_LM_DC_2ND_CLAMP6.Error_T2.STIME := T#0MS;
   S708_LM_DC_2ND_CLAMP6.Error_T2.ATIME := T#0MS;
   S708_LM_DC_2ND_CLAMP6.CHK_Aux1 := FALSE;
   S708_LM_DC_2ND_CLAMP6.CHK_Aux2 := FALSE;
   S708_LM_DC_2ND_CLAMP6.Error_T1_DN := FALSE;
   S708_LM_DC_2ND_CLAMP6.Error_T2_DN := FALSE;
   S708_LM_DC_2ND_CLAMP6.Adv_Memo := FALSE;
   S708_LM_DC_2ND_CLAMP6.Visu_Adv_Arr[0] := FALSE;
   S708_LM_DC_2ND_CLAMP6.Visu_Adv_Arr[1] := FALSE;
   S708_LM_DC_2ND_CLAMP6.Visu_Adv_Arr[2] := FALSE;
   S708_LM_DC_2ND_CLAMP6.Visu_Adv_Arr[3] := FALSE;
   S708_LM_DC_2ND_CLAMP6.Visu_Adv_Arr[4] := FALSE;
   S708_LM_DC_2ND_CLAMP6.Visu_Adv_Arr[5] := FALSE;
   S708_LM_DC_2ND_CLAMP6.Visu_Adv_Arr[6] := FALSE;
   S708_LM_DC_2ND_CLAMP6.Visu_Adv_Arr[7] := FALSE;
   S708_LM_DC_2ND_CLAMP6.Visu_Adv_Arr[8] := FALSE;
   S708_LM_DC_2ND_CLAMP6.Visu_Adv_Arr[9] := FALSE;
   S708_LM_DC_2ND_CLAMP6.Visu_Adv_Arr[10] := FALSE;
   S708_LM_DC_2ND_CLAMP6.Visu_Adv_Arr[11] := FALSE;
   S708_LM_DC_2ND_CLAMP6.Visu_Adv_Arr[12] := FALSE;
   S708_LM_DC_2ND_CLAMP6.Visu_Adv_Arr[13] := FALSE;
   S708_LM_DC_2ND_CLAMP6.Visu_Adv_Arr[14] := FALSE;
   S708_LM_DC_2ND_CLAMP6.Visu_Adv_Arr[15] := FALSE;
   S708_LM_DC_2ND_CLAMP6.Visu_Ret_Arr[0] := FALSE;
   S708_LM_DC_2ND_CLAMP6.Visu_Ret_Arr[1] := FALSE;
   S708_LM_DC_2ND_CLAMP6.Visu_Ret_Arr[2] := FALSE;
   S708_LM_DC_2ND_CLAMP6.Visu_Ret_Arr[3] := FALSE;
   S708_LM_DC_2ND_CLAMP6.Visu_Ret_Arr[4] := FALSE;
   S708_LM_DC_2ND_CLAMP6.Visu_Ret_Arr[5] := FALSE;
   S708_LM_DC_2ND_CLAMP6.Visu_Ret_Arr[6] := FALSE;
   S708_LM_DC_2ND_CLAMP6.Visu_Ret_Arr[7] := FALSE;
   S708_LM_DC_2ND_CLAMP6.Visu_Ret_Arr[8] := FALSE;
   S708_LM_DC_2ND_CLAMP6.Visu_Ret_Arr[9] := FALSE;
   S708_LM_DC_2ND_CLAMP6.Visu_Ret_Arr[10] := FALSE;
   S708_LM_DC_2ND_CLAMP6.Visu_Ret_Arr[11] := FALSE;
   S708_LM_DC_2ND_CLAMP6.Visu_Ret_Arr[12] := FALSE;
   S708_LM_DC_2ND_CLAMP6.Visu_Ret_Arr[13] := FALSE;
   S708_LM_DC_2ND_CLAMP6.Visu_Ret_Arr[14] := FALSE;
   S708_LM_DC_2ND_CLAMP6.Visu_Ret_Arr[15] := FALSE;
   S708_LM_DC_2ND_CLAMP6.BLK_Move_Ret := 0;
   S708_LM_DC_2ND_CLAMP6.Enable := FALSE;
   S708_LM_DC_2ND_CLAMP6.Adv_End := FALSE;
   S708_LM_DC_2ND_CLAMP6.Ret_End := FALSE;
   S708_LM_DC_2ND_CLAMP7.Enable_Aux := FALSE;
   S708_LM_DC_2ND_CLAMP7.Adv_Amount := 1;
   S708_LM_DC_2ND_CLAMP7.Ret_Amount := 1;
   S708_LM_DC_2ND_CLAMP7.LS_Adv1 := FALSE;
   S708_LM_DC_2ND_CLAMP7.LS_Ret1 := FALSE;
   S708_LM_DC_2ND_CLAMP7.LS_Adv2 := FALSE;
   S708_LM_DC_2ND_CLAMP7.LS_Ret2 := FALSE;
   S708_LM_DC_2ND_CLAMP7.LS_Adv3 := FALSE;
   S708_LM_DC_2ND_CLAMP7.LS_Ret3 := FALSE;
   S708_LM_DC_2ND_CLAMP7.LS_Adv4 := FALSE;
   S708_LM_DC_2ND_CLAMP7.LS_Ret4 := FALSE;
   S708_LM_DC_2ND_CLAMP7.SOL_Adv := FALSE;
   S708_LM_DC_2ND_CLAMP7.SOL_Ret := FALSE;
   S708_LM_DC_2ND_CLAMP7.M_Ready := TRUE;
   S708_LM_DC_2ND_CLAMP7.T_CHK1 := T#4S;
   S708_LM_DC_2ND_CLAMP7.T_CHK2 := T#4S;
   S708_LM_DC_2ND_CLAMP7.PB_Lamp_CHK := FALSE;
   S708_LM_DC_2ND_CLAMP7.PB_Error_Rst := FALSE;
   S708_LM_DC_2ND_CLAMP7.M_FLICK := TRUE;
   S708_LM_DC_2ND_CLAMP7.M_Adv_Err := FALSE;
   S708_LM_DC_2ND_CLAMP7.M_Ret_Err := FALSE;
   S708_LM_DC_2ND_CLAMP7.LP_Adv := FALSE;
   S708_LM_DC_2ND_CLAMP7.LP_Ret := FALSE;
   S708_LM_DC_2ND_CLAMP7.Visu_Adv := W#16#0;
   S708_LM_DC_2ND_CLAMP7.Visu_Ret := W#16#0;
   S708_LM_DC_2ND_CLAMP7.Error_T1.IN := FALSE;
   S708_LM_DC_2ND_CLAMP7.Error_T1.PT := T#4S;
   S708_LM_DC_2ND_CLAMP7.Error_T1.Q := FALSE;
   S708_LM_DC_2ND_CLAMP7.Error_T1.ET := T#0MS;
   S708_LM_DC_2ND_CLAMP7.Error_T1.STATE := B#16#0;
   S708_LM_DC_2ND_CLAMP7.Error_T1.STIME := T#22D23H1M2S541MS;
   S708_LM_DC_2ND_CLAMP7.Error_T1.ATIME := T#22D23H1M3S514MS;
   S708_LM_DC_2ND_CLAMP7.Error_T2.IN := FALSE;
   S708_LM_DC_2ND_CLAMP7.Error_T2.PT := T#4S;
   S708_LM_DC_2ND_CLAMP7.Error_T2.Q := FALSE;
   S708_LM_DC_2ND_CLAMP7.Error_T2.ET := T#0MS;
   S708_LM_DC_2ND_CLAMP7.Error_T2.STATE := B#16#0;
   S708_LM_DC_2ND_CLAMP7.Error_T2.STIME := T#0MS;
   S708_LM_DC_2ND_CLAMP7.Error_T2.ATIME := T#0MS;
   S708_LM_DC_2ND_CLAMP7.CHK_Aux1 := FALSE;
   S708_LM_DC_2ND_CLAMP7.CHK_Aux2 := FALSE;
   S708_LM_DC_2ND_CLAMP7.Error_T1_DN := FALSE;
   S708_LM_DC_2ND_CLAMP7.Error_T2_DN := FALSE;
   S708_LM_DC_2ND_CLAMP7.Adv_Memo := FALSE;
   S708_LM_DC_2ND_CLAMP7.Visu_Adv_Arr[0] := FALSE;
   S708_LM_DC_2ND_CLAMP7.Visu_Adv_Arr[1] := FALSE;
   S708_LM_DC_2ND_CLAMP7.Visu_Adv_Arr[2] := FALSE;
   S708_LM_DC_2ND_CLAMP7.Visu_Adv_Arr[3] := FALSE;
   S708_LM_DC_2ND_CLAMP7.Visu_Adv_Arr[4] := FALSE;
   S708_LM_DC_2ND_CLAMP7.Visu_Adv_Arr[5] := FALSE;
   S708_LM_DC_2ND_CLAMP7.Visu_Adv_Arr[6] := FALSE;
   S708_LM_DC_2ND_CLAMP7.Visu_Adv_Arr[7] := FALSE;
   S708_LM_DC_2ND_CLAMP7.Visu_Adv_Arr[8] := FALSE;
   S708_LM_DC_2ND_CLAMP7.Visu_Adv_Arr[9] := FALSE;
   S708_LM_DC_2ND_CLAMP7.Visu_Adv_Arr[10] := FALSE;
   S708_LM_DC_2ND_CLAMP7.Visu_Adv_Arr[11] := FALSE;
   S708_LM_DC_2ND_CLAMP7.Visu_Adv_Arr[12] := FALSE;
   S708_LM_DC_2ND_CLAMP7.Visu_Adv_Arr[13] := FALSE;
   S708_LM_DC_2ND_CLAMP7.Visu_Adv_Arr[14] := FALSE;
   S708_LM_DC_2ND_CLAMP7.Visu_Adv_Arr[15] := FALSE;
   S708_LM_DC_2ND_CLAMP7.Visu_Ret_Arr[0] := FALSE;
   S708_LM_DC_2ND_CLAMP7.Visu_Ret_Arr[1] := FALSE;
   S708_LM_DC_2ND_CLAMP7.Visu_Ret_Arr[2] := FALSE;
   S708_LM_DC_2ND_CLAMP7.Visu_Ret_Arr[3] := FALSE;
   S708_LM_DC_2ND_CLAMP7.Visu_Ret_Arr[4] := FALSE;
   S708_LM_DC_2ND_CLAMP7.Visu_Ret_Arr[5] := FALSE;
   S708_LM_DC_2ND_CLAMP7.Visu_Ret_Arr[6] := FALSE;
   S708_LM_DC_2ND_CLAMP7.Visu_Ret_Arr[7] := FALSE;
   S708_LM_DC_2ND_CLAMP7.Visu_Ret_Arr[8] := FALSE;
   S708_LM_DC_2ND_CLAMP7.Visu_Ret_Arr[9] := FALSE;
   S708_LM_DC_2ND_CLAMP7.Visu_Ret_Arr[10] := FALSE;
   S708_LM_DC_2ND_CLAMP7.Visu_Ret_Arr[11] := FALSE;
   S708_LM_DC_2ND_CLAMP7.Visu_Ret_Arr[12] := FALSE;
   S708_LM_DC_2ND_CLAMP7.Visu_Ret_Arr[13] := FALSE;
   S708_LM_DC_2ND_CLAMP7.Visu_Ret_Arr[14] := FALSE;
   S708_LM_DC_2ND_CLAMP7.Visu_Ret_Arr[15] := FALSE;
   S708_LM_DC_2ND_CLAMP7.BLK_Move_Ret := 0;
   S708_LM_DC_2ND_CLAMP7.Enable := FALSE;
   S708_LM_DC_2ND_CLAMP7.Adv_End := FALSE;
   S708_LM_DC_2ND_CLAMP7.Ret_End := FALSE;
   S708_LM_DC_1ST_CLAMP5.Enable_Aux := FALSE;
   S708_LM_DC_1ST_CLAMP5.Adv_Amount := 1;
   S708_LM_DC_1ST_CLAMP5.Ret_Amount := 1;
   S708_LM_DC_1ST_CLAMP5.LS_Adv1 := FALSE;
   S708_LM_DC_1ST_CLAMP5.LS_Ret1 := FALSE;
   S708_LM_DC_1ST_CLAMP5.LS_Adv2 := FALSE;
   S708_LM_DC_1ST_CLAMP5.LS_Ret2 := FALSE;
   S708_LM_DC_1ST_CLAMP5.LS_Adv3 := FALSE;
   S708_LM_DC_1ST_CLAMP5.LS_Ret3 := FALSE;
   S708_LM_DC_1ST_CLAMP5.LS_Adv4 := FALSE;
   S708_LM_DC_1ST_CLAMP5.LS_Ret4 := FALSE;
   S708_LM_DC_1ST_CLAMP5.SOL_Adv := FALSE;
   S708_LM_DC_1ST_CLAMP5.SOL_Ret := FALSE;
   S708_LM_DC_1ST_CLAMP5.M_Ready := TRUE;
   S708_LM_DC_1ST_CLAMP5.T_CHK1 := T#4S;
   S708_LM_DC_1ST_CLAMP5.T_CHK2 := T#4S;
   S708_LM_DC_1ST_CLAMP5.PB_Lamp_CHK := FALSE;
   S708_LM_DC_1ST_CLAMP5.PB_Error_Rst := FALSE;
   S708_LM_DC_1ST_CLAMP5.M_FLICK := TRUE;
   S708_LM_DC_1ST_CLAMP5.M_Adv_Err := FALSE;
   S708_LM_DC_1ST_CLAMP5.M_Ret_Err := FALSE;
   S708_LM_DC_1ST_CLAMP5.LP_Adv := FALSE;
   S708_LM_DC_1ST_CLAMP5.LP_Ret := FALSE;
   S708_LM_DC_1ST_CLAMP5.Visu_Adv := W#16#0;
   S708_LM_DC_1ST_CLAMP5.Visu_Ret := W#16#0;
   S708_LM_DC_1ST_CLAMP5.Error_T1.IN := FALSE;
   S708_LM_DC_1ST_CLAMP5.Error_T1.PT := T#4S;
   S708_LM_DC_1ST_CLAMP5.Error_T1.Q := FALSE;
   S708_LM_DC_1ST_CLAMP5.Error_T1.ET := T#0MS;
   S708_LM_DC_1ST_CLAMP5.Error_T1.STATE := B#16#0;
   S708_LM_DC_1ST_CLAMP5.Error_T1.STIME := T#22D23H1M3S514MS;
   S708_LM_DC_1ST_CLAMP5.Error_T1.ATIME := T#22D23H1M3S968MS;
   S708_LM_DC_1ST_CLAMP5.Error_T2.IN := FALSE;
   S708_LM_DC_1ST_CLAMP5.Error_T2.PT := T#4S;
   S708_LM_DC_1ST_CLAMP5.Error_T2.Q := FALSE;
   S708_LM_DC_1ST_CLAMP5.Error_T2.ET := T#0MS;
   S708_LM_DC_1ST_CLAMP5.Error_T2.STATE := B#16#0;
   S708_LM_DC_1ST_CLAMP5.Error_T2.STIME := T#0MS;
   S708_LM_DC_1ST_CLAMP5.Error_T2.ATIME := T#0MS;
   S708_LM_DC_1ST_CLAMP5.CHK_Aux1 := FALSE;
   S708_LM_DC_1ST_CLAMP5.CHK_Aux2 := FALSE;
   S708_LM_DC_1ST_CLAMP5.Error_T1_DN := FALSE;
   S708_LM_DC_1ST_CLAMP5.Error_T2_DN := FALSE;
   S708_LM_DC_1ST_CLAMP5.Adv_Memo := FALSE;
   S708_LM_DC_1ST_CLAMP5.Visu_Adv_Arr[0] := FALSE;
   S708_LM_DC_1ST_CLAMP5.Visu_Adv_Arr[1] := FALSE;
   S708_LM_DC_1ST_CLAMP5.Visu_Adv_Arr[2] := FALSE;
   S708_LM_DC_1ST_CLAMP5.Visu_Adv_Arr[3] := FALSE;
   S708_LM_DC_1ST_CLAMP5.Visu_Adv_Arr[4] := FALSE;
   S708_LM_DC_1ST_CLAMP5.Visu_Adv_Arr[5] := FALSE;
   S708_LM_DC_1ST_CLAMP5.Visu_Adv_Arr[6] := FALSE;
   S708_LM_DC_1ST_CLAMP5.Visu_Adv_Arr[7] := FALSE;
   S708_LM_DC_1ST_CLAMP5.Visu_Adv_Arr[8] := FALSE;
   S708_LM_DC_1ST_CLAMP5.Visu_Adv_Arr[9] := FALSE;
   S708_LM_DC_1ST_CLAMP5.Visu_Adv_Arr[10] := FALSE;
   S708_LM_DC_1ST_CLAMP5.Visu_Adv_Arr[11] := FALSE;
   S708_LM_DC_1ST_CLAMP5.Visu_Adv_Arr[12] := FALSE;
   S708_LM_DC_1ST_CLAMP5.Visu_Adv_Arr[13] := FALSE;
   S708_LM_DC_1ST_CLAMP5.Visu_Adv_Arr[14] := FALSE;
   S708_LM_DC_1ST_CLAMP5.Visu_Adv_Arr[15] := FALSE;
   S708_LM_DC_1ST_CLAMP5.Visu_Ret_Arr[0] := FALSE;
   S708_LM_DC_1ST_CLAMP5.Visu_Ret_Arr[1] := FALSE;
   S708_LM_DC_1ST_CLAMP5.Visu_Ret_Arr[2] := FALSE;
   S708_LM_DC_1ST_CLAMP5.Visu_Ret_Arr[3] := FALSE;
   S708_LM_DC_1ST_CLAMP5.Visu_Ret_Arr[4] := FALSE;
   S708_LM_DC_1ST_CLAMP5.Visu_Ret_Arr[5] := FALSE;
   S708_LM_DC_1ST_CLAMP5.Visu_Ret_Arr[6] := FALSE;
   S708_LM_DC_1ST_CLAMP5.Visu_Ret_Arr[7] := FALSE;
   S708_LM_DC_1ST_CLAMP5.Visu_Ret_Arr[8] := FALSE;
   S708_LM_DC_1ST_CLAMP5.Visu_Ret_Arr[9] := FALSE;
   S708_LM_DC_1ST_CLAMP5.Visu_Ret_Arr[10] := FALSE;
   S708_LM_DC_1ST_CLAMP5.Visu_Ret_Arr[11] := FALSE;
   S708_LM_DC_1ST_CLAMP5.Visu_Ret_Arr[12] := FALSE;
   S708_LM_DC_1ST_CLAMP5.Visu_Ret_Arr[13] := FALSE;
   S708_LM_DC_1ST_CLAMP5.Visu_Ret_Arr[14] := FALSE;
   S708_LM_DC_1ST_CLAMP5.Visu_Ret_Arr[15] := FALSE;
   S708_LM_DC_1ST_CLAMP5.BLK_Move_Ret := 0;
   S708_LM_DC_1ST_CLAMP5.Enable := FALSE;
   S708_LM_DC_1ST_CLAMP5.Adv_End := FALSE;
   S708_LM_DC_1ST_CLAMP5.Ret_End := FALSE;
END_DATA_BLOCK

FUNCTION FC 143 : VOID
TITLE =
NAME : DAECHA
VERSION : 0.1

BEGIN
NETWORK
TITLE =
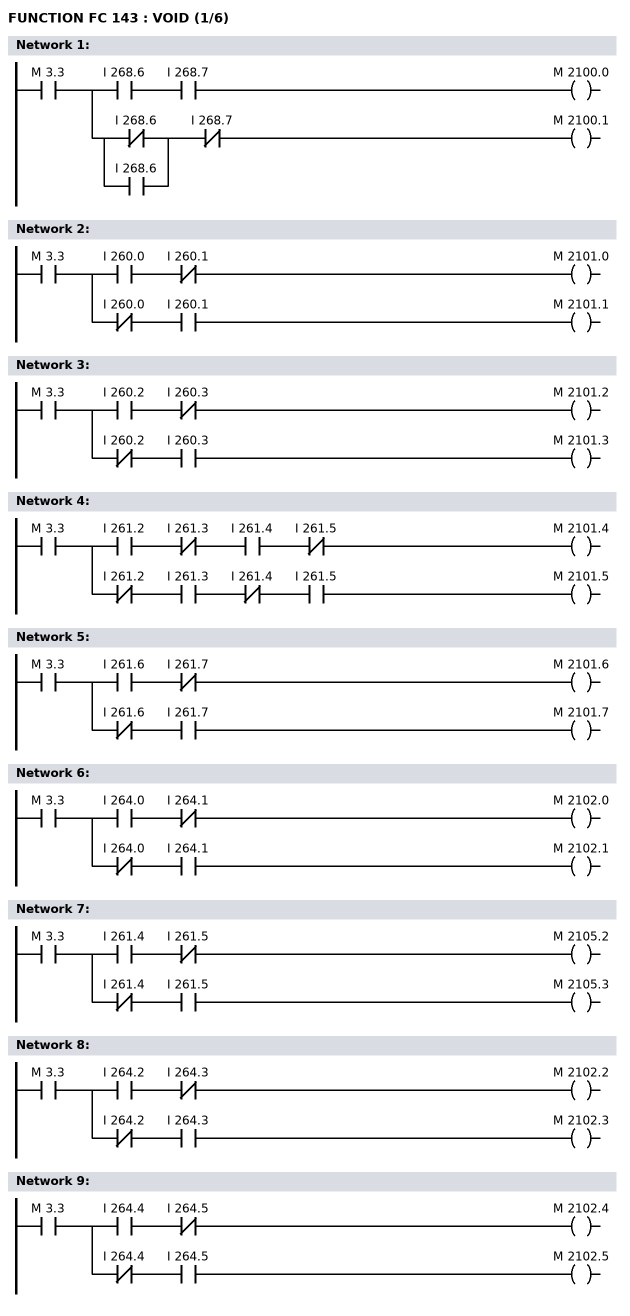

      A     M      3.3;
      =     L      0.0;
      A     L      0.0;
      A     I    268.6;
      A     I    268.7;
      =     M   2100.0;
      A     L      0.0;
      A(    ;
      ON    I    268.6;
      O     I    268.6;
      )     ;
      AN    I    268.7;
      =     M   2100.1;
NETWORK
TITLE =

      A     M      3.3;
      =     L      0.0;
      A     L      0.0;
      A     I    260.0;
      AN    I    260.1;
      =     M   2101.0;
      A     L      0.0;
      AN    I    260.0;
      A     I    260.1;
      =     M   2101.1;
NETWORK
TITLE =

      A     M      3.3;
      =     L      0.0;
      A     L      0.0;
      A     I    260.2;
      AN    I    260.3;
      =     M   2101.2;
      A     L      0.0;
      AN    I    260.2;
      A     I    260.3;
      =     M   2101.3;
NETWORK
TITLE =

      A     M      3.3;
      =     L      0.0;
      A     L      0.0;
      A     I    261.2;
      AN    I    261.3;
      A     I    261.4;
      AN    I    261.5;
      =     M   2101.4;
      A     L      0.0;
      AN    I    261.2;
      A     I    261.3;
      AN    I    261.4;
      A     I    261.5;
      =     M   2101.5;
NETWORK
TITLE =

      A     M      3.3;
      =     L      0.0;
      A     L      0.0;
      A     I    261.6;
      AN    I    261.7;
      =     M   2101.6;
      A     L      0.0;
      AN    I    261.6;
      A     I    261.7;
      =     M   2101.7;
NETWORK
TITLE =

      A     M      3.3;
      =     L      0.0;
      A     L      0.0;
      A     I    264.0;
      AN    I    264.1;
      =     M   2102.0;
      A     L      0.0;
      AN    I    264.0;
      A     I    264.1;
      =     M   2102.1;
NETWORK
TITLE =

      A     M      3.3;
      =     L      0.0;
      A     L      0.0;
      A     I    261.4;
      AN    I    261.5;
      =     M   2105.2;
      A     L      0.0;
      AN    I    261.4;
      A     I    261.5;
      =     M   2105.3;
NETWORK
TITLE =

